(* CODESYS project Raspberry I2C MUX.library
   Author: Stefan Dreyer
   Version: 1.0.1.1
   Description: Library containing device support for different I2C slaves under Raspberry Pi with multiplexer Support
      
      Using some cool function of OSCAT library.
      look at www.oscat.de
   Title: Raspberry I2C MUX
   DefaultNamespace: I2C_MUX
   Company: Stefan Dreyer

Project tree, tasks and I/O mapping:
  libraries: IoStandard, * (System); Standard, * (System); Time and Date, 3.5.7.0 (3S - Smart Software Solutions GmbH); BUILDING, 1.0.0.0 (OSCAT); VisuDialogs, * (System); BASIC, 3.3.3.0 (OSCAT); CAA Memory, 3.5.12.0 (CAA Technical Workgroup); Common Helper for development, 1.0.0.0 (Stefan Dreyer); Raspberry Pi Peripherals, 3.5.13.0 (3S - Smart Software Solutions GmbH); SysSem, 3.5.15.0 (System)
  00000000-0000-0000-0000-000000000000|D:\CoDeSys\LibrariesV3\trunk\Intern\CAA\CAA Template\3.4.0.0 draft\Placeholder.xml
  00000000-0000-0000-0000-000000000000|D:\CoDeSys\LibrariesV3\trunk\Intern\CAA\CAA Template\3.2.0.3 draft\Prefix.pdf
  00000000-0000-0000-0000-000000000000|D:\CoDeSys\LibrariesV3\trunk\Intern\CAA\CAA Template\3.5.2.0 draft\Placeholder.xml
  global variables GVL
  Externe Datei
  Structs/
    data type BusCycleTime
    data type requestData
    data type BME280Data
    data type MUX_COM
    data type SOFT_FONT_DATA
    data type SI7021Data
    data type BMP280Data
  GlobalConstants/
    global variables MyConstants
  Function Blocks/
    function block TCA9548 [ST]: Initialize, BeforeWriteOutputs, goError, BIT_OF_BYTE, restartBus, checkRequestChange, getFirstDifferentStage, clearUnnededStages, setStages
    function block PCA9555OUT [ST]: Initialize, BeforeWriteOutputs
    function block PCA9555IN [ST]: Initialize, AfterReadInputs
    function block BME280 [ST]: AfterReadInputs, Initialize, BeforeWriteOutputs, initCalibration, initDevice, setForcedMode, calcControlRegister
    function block I2C_BASE [ST]: Initialize, AfterReadInputs, BeforeWriteOutputs, checkWrite, checkWrite8, checkReadRegister, goError, checkMultiplex, resetSysCallNum, checkWriteTimeMultiplex, checkReadTimeMultiplex, checkInitMultiplex, checkSet, setRequest, checkMasterFree, resetRequest, checkDeviceOnError, calcCycleTime, checkRead, DeviceState, DeviceRunning
    function block TSL2561 [ST]: AfterReadInputs, Initialize, BeforeWriteOutputs, initDevice, checkDevice, writeControlRegister, setCommandRegister, startDevice, stopDevice, getData, calculateLux
    function block PCF8575IN [ST]: Initialize, AfterReadInputs
    function block PCA9685 [ST]: BeforeWriteOutputs, Initialize, calcOut
    function block Dim4Ch [ST]: BeforeWriteOutputs, Initialize, calcOut
    function block EEPROM_24C512 [ST]: Initialize, AfterReadInputs, BeforeWriteOutputs
    function block SSD1306 [ST]: Initialize, BeforeWriteOutputs, DisplayOn, DisplayOff, SetCommand, SetContrast, DrawLine, SetPixelCache, GetCacheByte, SetCacheByteRaw, WriteCacheToLcd, SetByteCache, SetSoftFont, WriteChar, FillBox, LineFeed, SetCursor
    function block PCF8575OUT [ST]: Initialize, BeforeWriteOutputs
    function block SI7021 [ST]: AfterReadInputs, BeforeWriteOutputs, Initialize
    function block BMP280 [ST]: AfterReadInputs, Initialize, BeforeWriteOutputs, initCalibration, initDevice, setForcedMode, calcControlRegister
  VISU/
    visualisation SSD1306
  text list GlobalTextList
  ENUMS/
    data type LCD_MODES
    data type SOFT_FONT_NUMS
  TextLists/
    text list SOFT_FONT_NAMES
*)

// Structs/BusCycleTime
TYPE BusCycleTime :
STRUCT
	//Cycle Time in ms
	cycleTime:UDINT;
	//last tick for cycle Time
	cycleTimeLastTick:CAA.TICK;
	//cycle frequency 
	cycleFrequency:LREAL;
END_STRUCT
END_TYPE

// Structs/requestData
TYPE requestData :
STRUCT
	//time to next acions
	varTime: CAA.TICK;
	//request var by child outside time, only internal use
	varRequest: BOOL;
	//time between actions in ms
	timePreset:UDINT;
	//set to request by child
	request : BOOL := FALSE;
	//cycle Time of this request
	cycleTime:BusCycleTime;
END_STRUCT
END_TYPE

// Structs/BME280Data
TYPE BME280Data :
STRUCT
	//Possible Data from BME280 from Bosch Sensor Tec
	//using -->LREAL;
	Temperatur:LREAL;//using -->LREAL;
	//using -->LREAL;
	Humidity:LREAL;//using -->LREAL;
	//using -->LREAL;
	Pressure: LREAL;//using -->LREAL;
	//using -->REAL;
	absHumidity:REAL;//using -->REAL;
	//using -->REAL;
	dewPoint:REAL;//using -->REAL;

	(*
		//using -->LREAL;
	Temperatur:CommonTypes.ALL_TYPES_UNION;//using -->LREAL;
	//using -->LREAL;
	Humidity:CommonTypes.ALL_TYPES_UNION;//using -->LREAL;
	//using -->LREAL;
	Pressure: CommonTypes.ALL_TYPES_UNION;//using -->LREAL;
	//using -->REAL;
	absHumidity:CommonTypes.ALL_TYPES_UNION;//using -->REAL;
	//using -->REAL;
	dewPoint:CommonTypes.ALL_TYPES_UNION;//using -->REAL
	*)
	
END_STRUCT
END_TYPE

// Structs/MUX_COM
TYPE MUX_COM :
STRUCT
	
	//Call Number, Order by system call
	callNum:UINT:=0;
	//Start Read differenz for unload cycle load
	//startReadDifferenz:UDINT;
	//muxNum of which slave multiplexer is dead
	//muxNumDead:INT;
	//set this to restart the bus
	startRestartBus: BOOL;

	//set when "last" multiplexer detect to restart the bus
	restartBus: BOOL;
	

	//is init after multiplexer error, all multiplex slaves have to be off
	initAfterError: BOOL;
	//multiplex numbers requestet by on slave
	muxChannelRequest:ARRAY[0..7] OF USINT;
	//multiplex numbers set by master
	muxChannelSet:ARRAY[0..7] OF USINT;
	//instans number of fb who requestet the bus
	fbRequest: INT;

	//count of stages
	stages:UINT;
	//if set, value in stages is valid, so slaves can check there mux nums
	stagesValid: BOOL;
	//mux chain i.O.
	//chainIo:BOOL;
END_STRUCT
END_TYPE

// ENUMS/LCD_MODES
{attribute 'qualified_only'}
{attribute 'strict'}
TYPE LCD_MODES :
(
	CLEAR_BIT := 0, SET_BIT := 1, INVERT_BIT := 2 
)USINT;
END_TYPE

// ENUMS/SOFT_FONT_NUMS
{attribute 'qualified_only'}
{attribute 'strict'}
TYPE SOFT_FONT_NUMS :
(
	FONT_4X6 := 0, FONT_5X8 := 1, FONT_5X12 := 2, FONT_6X8 := 3, FONT_6X10 := 4, FONT_7X12 := 5,
	FONT_7X12B := 6, FONT_8X8 := 7, FONT_8X12 := 8, FONT_8X14 := 9,
	FONT_10X16 := 10, FONT_12X16 := 11, FONT_16X8 := 12,
	FONT_16X12 := 13, FONT_16X26 := 14, last := 15
)USINT;
END_TYPE

// Structs/SOFT_FONT_DATA
TYPE SOFT_FONT_DATA :
STRUCT
	width:USINT;
	height:USINT;
	mask:DWORD;
	data:POINTER TO BYTE;
	size:USINT;
END_STRUCT
END_TYPE

// Structs/SI7021Data
TYPE SI7021Data :
STRUCT
	//Possible Data from BME280 from Bosch Sensor Tec
	//using -->LREAL;
	Temperatur:LREAL;//using -->LREAL;
	//using -->LREAL;
	Humidity:LREAL;//using -->LREAL;
	//using -->REAL;
	absHumidity:REAL;//using -->REAL;
	//using -->REAL;
	dewPoint:REAL;//using -->REAL;

END_STRUCT
END_TYPE

// Structs/BMP280Data
TYPE BMP280Data :
STRUCT
	//Possible Data from BME280 from Bosch Sensor Tec
	//using -->LREAL;
	Temperatur:LREAL;//using -->LREAL;
	//using -->LREAL;
	Pressure: LREAL;//using -->LREAL;

	
END_STRUCT
END_TYPE

// GVL
{attribute 'qualified_only'}
VAR_GLOBAL
	MUX_COMS:ARRAY[0..7]OF MUX_COM;

END_VAR
VAR_GLOBAL CONSTANT
	PCA9685_MODE1: USINT := 0;
	PCA9685_MODE2: USINT := 1;
	PCA9685_PRESCALE: USINT := 16#FE;
	
	LED0_ON_L: USINT := 16#6;
	LED0_ON_H: USINT := 16#7;
	LED0_OFF_L: USINT := 16#8;
	LED0_OFF_H: USINT := 16#9;
END_VAR

// GlobalConstants/MyConstants
{attribute 'qualified_only'}
VAR_GLOBAL CONSTANT

				
END_VAR

// Function Blocks/TCA9548

(*
Function for i2c Multiplexer
so all new, yeha!!!
the slave are requesting an connection to there hardware and writing the channel numbers(of TCA9548) corospending on the hardware in the request array.
and so the master trys to deliver. he checks if a part of the request is already suitable and changes the rest if not.
on init the master tells the slaves how much stages ar avalibel, and so the the slave can check if there config is i.O.
if there are to much stages in the config, the slaves go in error(TODO!!!)
convention: a slave doesn't set a request if the actuel Multiplex set suits his communication request also partially
*)
FUNCTION_BLOCK TCA9548 EXTENDS I2C_BASE

VAR

	stageAddresses:ARRAY[0..7] OF USINT;
	//count of vailid stages
	stages:UINT;
	//which stage ist the last actually
	actLastStage:INT;
	
	outMask:ARRAY[0..7] OF BYTE := [2#1, 2#10, 2#100, 2#1000, 2#10000, 2#100000, 2#1000000, 2#10000000];
	
	//how often i have to try bevor i know i am dead
	retryCountPreload:UINT;
	//var for count trying
	retryCount:UINT;
END_VAR

VAR CONSTANT 
	DEAD_DEVICE:INT:=100;
END_VAR

SUPER^();

METHOD Initialize : UDINT
VAR_INPUT
	wModuleType : UINT;
	dwInstance : UDINT;
	pConnector : POINTER TO IoConfigConnector;
END_VAR
VAR
	pParam: POINTER TO IoConfigParameter;		
	udiResult: UDINT;
 	i:INT;
	iPointer:POINTER TO usINT;
	pLength:DWORD;
END_VAR
SUPER^.Initialize(wModuleType, dwInstance, pConnector);


pParam := ConfigGetParameter(_pConnector, 20);
retryCountPreload := IoStandard.ConfigGetParameterValueWord(pParam, ADR(udiResult));

pParam := ConfigGetParameter(_pConnector, 21);
iPointer := IoStandard.ConfigGetParameterValuePointer(pParam, ADR(udiResult)); 
pLength := IoStandard.ConfigGetParameterLength(pParam);

//copy addresses to instance var
FOR i := 0 TO DWORD_TO_INT(pLength) / 8 DO
	stageAddresses[i+1] := iPointer[i];
END_FOR
//set first stage address in array
stageAddresses[0] := usiAddress;
pParam := ConfigGetParameter(_pConnector, 22);
stages := IoStandard.ConfigGetParameterValueWord(pParam, ADR(udiResult));
GVL.MUX_COMS[numMuxMaster].stages := stages;

GVL.MUX_COMS[numMuxMaster].stagesValid := TRUE;

//actLastStage := 1;

stateAfterError := RETRY_DEVICE;
stateAfterInit := RUN_DEVICE;
//don't use step ERROR_DEVICE in super FB
stateOnError := RETRY_DEVICE;
//GVL.MUX_COMS[numMuxMaster].chainIo := TRUE;
END_METHOD

METHOD BeforeWriteOutputs : INT
VAR
	firstDifferentStage: INT;
	returnByte: BYTE;
END_VAR
SUPER^.BeforeWriteOutputs();

CASE _iState OF

	RUN_DEVICE:
	//hello again folks! i am glad to see you on my next experiment
	//Multiplexing I2C with request from slaves, so lets do it
	IF checkRequestChange() THEN//gotcha, something to do...
		firstDifferentStage := getFirstDifferentStage();
		//if first different in request = 0 then the set have to be resetet from aktStage to Stage 1
		//stage 0 don't need to be cleard, because it is overriden 
		IF actLastStage > firstDifferentStage THEN
			IF clearUnnededStages(firstDifferentStage) = ERROR_RET_VAL THEN
				//error on clear multiplexer
				RETURN;
			END_IF
		END_IF
		IF setStages(firstDifferentStage)  = ERROR_RET_VAL THEN
			RETURN;
		END_IF
	END_IF
 	GVL.MUX_COMS[numMuxMaster].initAfterError := FALSE;
	RETRY_DEVICE:
	IF checkRead(pbyBuffer:= ADR(returnByte), nBufferLen:= 1)  = READ_SUCCSESSFULL THEN
		_iState := RUN_DEVICE;
	END_IF
	//GVL.MUX_COMS[numMuxMaster].chainIo := TRUE;
	
	DEAD_DEVICE:
	//here we can do just nothing ...
	//or wait for an restart from main cycle ...

END_CASE
END_METHOD

METHOD goError
VAR_INPUT
	ReadWrite:BOOL;
END_VAR
VAR
	i:INT;
END_VAR
IF _iState = RUN_DEVICE THEN
	retryCount := retryCountPreload;
END_IF
SUPER^.goError(ReadWrite := FALSE);

//GVL.MUX_COMS[numMuxMaster].chainIo := FALSE;
GVL.MUX_COMS[numMuxMaster].initAfterError := TRUE;
//reset all requests and stages
FOR i := 0 TO  STAGES_END DO
	GVL.MUX_COMS[numMuxMaster].muxChannelSet[i]:= 0;
	GVL.MUX_COMS[numMuxMaster].muxChannelRequest[i]:=0;
END_FOR
END_METHOD

METHOD BIT_OF_BYTE : bool
VAR_INPUT

	in : BYTE;
	N : INT;

END_VAR
BIT_OF_BYTE := (SHR(in,N) AND 16#00000001) > 0;
END_METHOD

//call this from main PUO for try to restart the bus
METHOD restartBus
VAR_INPUT


END_VAR
GVL.MUX_COMS[numMuxMaster].startRestartBus := TRUE;
END_METHOD

METHOD checkRequestChange : bool
VAR_INPUT
END_VAR
VAR
	i:uINT;
END_VAR
//checking if the master have something to to...
checkRequestChange := FALSE;
FOR i := 0 TO stages DO
	IF GVL.MUX_COMS[numMuxMaster].muxChannelRequest[i] <> 0 THEN
		checkRequestChange := TRUE;
	END_IF
END_FOR
END_METHOD

METHOD getFirstDifferentStage : int
VAR_INPUT
END_VAR
VAR
	i:int;	
END_VAR
getFirstDifferentStage := 0;

FOR i := 0 TO 7 DO
	IF GVL.MUX_COMS[numMuxMaster].muxChannelRequest[i] <> GVL.MUX_COMS[numMuxMaster].muxChannelSet[i] THEN
		//it have to hit at interation 7 else a slvae has set an request 
		//for an excisting set
		getFirstDifferentStage := i;
		RETURN;
	END_IF
END_FOR
END_METHOD

METHOD clearUnnededStages : INT
VAR_INPUT
	firstDifferentStage:INT;
	
END_VAR
VAR
	byteBuffer:ARRAY[0..0] OF BYTE;
	i:INT;
	writeRetVal:DINT;
END_VAR
clearUnnededStages := WRITE_SUCCSESSFULL;
//my clear byte
byteBuffer[0] := 0;
FOR i := actLastStage TO firstDifferentStage + 1 BY -1  DO
	//write here with master write
	writeRetVal := _pMaster^.write(stageAddresses[i],ADR(byteBuffer),1);
	IF writeRetVal <> 1 AND NOT debugSlave THEN
		//SUPER^.goError();
		goError(ReadWrite := FALSE);
		clearUnnededStages := ERROR_RET_VAL;
		RETURN;  
	END_IF
	//did go one stage back
	actLastStage := i - 1;
	//and set set
	GVL.MUX_COMS[numMuxMaster].muxChannelSet[i] := 0;
END_FOR
END_METHOD

METHOD setStages : int
VAR_INPUT
	firstDifferentStage:INT;
END_VAR
VAR
	i:INT;
	writeRetVal: DINT;
	byteBuffer: array[0..0] of byte;
END_VAR
setStages := WRITE_SUCCSESSFULL;
FOR i := firstDifferentStage TO 7 DO
	IF GVL.MUX_COMS[numMuxMaster].muxChannelRequest[i] = 0 THEN
		RETURN;//everything done
	END_IF
	byteBuffer[0] := outMask[GVL.MUX_COMS[numMuxMaster].muxChannelRequest[i]-1];
	writeRetVal := _pMaster^.write(stageAddresses[i],ADR(byteBuffer),1);
	IF writeRetVal <> 1 AND NOT debugSlave THEN
		//SUPER^.goError();
		goError(ReadWrite := FALSE);
		setStages := ERROR_RET_VAL;
		RETURN;  
	END_IF
	//set stage set
	GVL.MUX_COMS[numMuxMaster].muxChannelSet[i] := GVL.MUX_COMS[numMuxMaster].muxChannelRequest[i];
	//did go one stage forward
	actLastStage := i;
END_FOR
END_METHOD

END_FUNCTION_BLOCK

// Function Blocks/I2C_BASE
(*Multiplex howto

one I2C_BASE FB is createt by an derive of 3s class i2c

in this fb all Multiplex stuff an controlling Stuff of an i2c slave is beeing done.

childs of this base FB must call parent methods, if theys use and hide the parent method.

the Multiplexing is Programmend for an TCA9548 chip,

you can combinie this chips until the adresses are empty... 

so you can cascade them, or use 8 of them parallel

or 4 parallel an cascade after them, just take care that the adresses can't collid.

in the device descripten the option MUX_MASTER calls the slave behinde which slave they are. It allthow tells the muxer which "row" he serves.

If you cascade the Muxers you don't need to da them in the device tree. the first muxer programm does the stuff for the cascaded ones. so you have to tell the first muxer in the device description,

on which stage after him which adress auf the muxers is being used

So this might an bit confusing, but i did it so ...

So every slave behind an muxer have to tell the master behind which channes of the muxer(s) he is, if he want to communicate.

So you have to see which slaves you do far behinde the pi, because the shold communicate least.

If you have some IO which have to be fast, put them near to the pi

If you have may an io expander with 8 adressesw free, put them behinde one muxer an you can use 8*8 = 64 aof them. ist they are 16 bit then it is 1024 io's

Else, put 8 muxer behinde one muxer and you have 8*8*8*16=8192 IOs. and this with only 9 muxers :D. and 512 IO chips ...

So take care how often the muxed slaves want to communicate because each time the muxer have to be switched.

Allthow you can tell the slaves that they can use foreign requests. This means, if the ar 3 devices behinde on mux channel(don't care aboute the position in the row) and one does request an communication,

The slaves with activatet foreign request do allthow communicatet an reset here own timer. So you can reduse the muxing switching bus load.

You althow cann tell the salve how often they have to communicate, do this in the device description, an look to the exampel devices. 

You althow can request an communication without the timer. Maybe on if an output have changed or you recived an interrupt for an I2C slave.

Look to dhe devices i have used it a some times.

Hi Zdenko,

you need to change this in:

/etc/init.d/codesyscontrol 

snippet:

Code:

        make_mknod

        killall codesyscontrol.bin > /dev/null;

        export PlcConfigFile=/etc/CODESYSControl.cfg

        echo bcm2708_i2c.0 > /sys/bus/platform/drivers/bcm2708_i2c/unbind
        echo 400000 > /sys/module/i2c_bcm2708/parameters/baudrate
        echo bcm2708_i2c.0 > /sys/bus/platform/drivers/bcm2708_i2c/bind




*)
FUNCTION_BLOCK I2C_BASE EXTENDS i2c
VAR_IN_OUT
	
END_VAR

VAR_OUTPUT

	RETVAL:DINT;
	ERROR: BOOL;
	TimeOutHit:BOOL;

END_VAR
VAR
	i:UINT;
	//slave is behind an multiplexer
	isMultiplex: BOOL;
	
 	stageChannelNums:ARRAY[0..STAGES_END] OF USINT;
	//if set use a foreign request to communicate
	useForeign: BOOL;
	//set if an request is set by myself for read
	//requestRead: BOOL;
	//set if an request is set by myself for write
	//requestWrite: BOOL;

	//state auf state maschine after an erre, change on your needs in initialisize
	stateAfterError:INT:=START_INIT;
	stateAfterInit:INT:=START_INIT;
	stateOnError:INT := ERROR_DEVICE;
	
	countNextTry:UDINT;

	waitAfterFault: BOOL;
	cyclseToWaitAfterFault:UDINT:=100;
	
	errorFromChild: BOOL := FALSE;
	

	// Call Number in Order of System call
	sysCallNumRead: UINT;
	sysCallNumWrite: UINT;
	
	readAttempts:LINT;
	writeAttempts:LINT;
	//is Read function called?
	didRead: BOOL := FALSE;
	//is write fucntion called?
	didWrite: BOOL := FALSE;
	//have i to report device i.o.?
	debugSlave: BOOL;
	//request data for read
	readRequest:requestData;
 	//request data for write
	writeRequest:requestData;
	
	numMuxMaster:USINT;
 
	ErrorCountRead:ULINT;
	ErrorCountWrite:ULINT;
	TimeOut:ton;

	
END_VAR
VAR_TEMP	

END_VAR

VAR CONSTANT 

STAGES_END:INT:=7;	

ERROR_DEVICE:INT:=40;
ERROR_RET_VAL:INT:=-1;
WRITE_SUCCSESSFULL:INT:=1;
READ_SUCCSESSFULL:INT:=2;
CHECK_SET_IO:INT:=1;

START_INIT:INT:=5;
WAIT_FOR_STAGES:INT:=1;
START_DEVICE:INT:=6;
RUN_DEVICE:INT:=10;
RETRY_DEVICE:INT:=20;
WAIT_DEVICE:INT:=30;

END_VAR

SUPER^();

(*
try to call this only once per cycle
but it is called by AfterReadInputs an BeforWriteOutputs
so try to check if both function are called by device description 
and if both activ do at read and else in the function called allone

*)
TimeOut(IN := _iState <> 10, PT:=T#1S, Q=> TimeOutHit);

IF _xAfterReadInputs = FALSE AND didRead AND didWrite THEN
	RETURN;
END_IF

//check if mux master gone erre, if so, go self to error
IF checkInitMultiplex() THEN
	goError(ReadWrite := TRUE);
END_IF
 

CASE _iState OF
0:
	IF isMultiplex THEN
		_iState := WAIT_FOR_STAGES;
	ELSE
		_iState := stateAfterInit;
	END_IF
WAIT_FOR_STAGES:
	IF GVL.MUX_COMS[numMuxMaster].stagesValid THEN
		//check muxnums deap
		//if to much muxnums ... error
		FOR i := 0 TO INT_TO_UINT(STAGES_END) DO
			IF stageChannelNums[i] <> 0 AND GVL.MUX_COMS[numMuxMaster].stages < i THEN
				_iState := WAIT_DEVICE;
				
				RETURN;
			END_IF
		END_FOR
		_iState := stateAfterInit;
	END_IF

ERROR_DEVICE:
	IF NOT waitAfterFault THEN
		_iState := stateAfterError;
	ELSE
		IF countNextTry > 0 THEN
			countNextTry := countNextTry- 1;
		END_IF
		IF countNextTry = 0 THEN
			_iState := stateAfterError;
		END_IF
	END_IF
WAIT_DEVICE:
//wrong config, nothing to do
END_CASE


ERROR := _iState <> RUN_DEVICE OR errorFromChild;

METHOD Initialize : UDINT
VAR_INPUT
	wModuleType : UINT;
	dwInstance : UDINT;
	pConnector : POINTER TO IoConfigConnector;
END_VAR
VAR
	pParam: POINTER TO IoConfigParameter;		
	udiResult: UDINT;
	byte1:byte;
	siPointer: POINTER TO USINT;
	pLength: DWORD;
	i: INT;
END_VAR
SUPER^.Initialize(wModuleType, dwInstance, pConnector);
//make differez in start reading, very rudimentary

//MUX_COM.startReadDifferenz := MUX_COM.startReadDifferenz +1;

(*get Adress from config*)
pParam := ConfigGetParameter(_pConnector, 1);
usiAddress:= IoStandard.ConfigGetParameterValueByte(pParam, ADR(udiResult));


(*get status of is this Mutiplex adress*)
pParam := ConfigGetParameter(_pConnector, 2);
byte1:= IoStandard.ConfigGetParameterValueByte(pParam, ADR(udiResult));
IF byte1 = BYTE#1 THEN
	isMultiplex:=TRUE;
ELSE
	isMultiplex:=FALSE;	
END_IF


pParam := ConfigGetParameter(_pConnector, 3);
siPointer := IoStandard.ConfigGetParameterValuePointer(pParam, ADR(udiResult)); 
pLength := IoStandard.ConfigGetParameterLength(pParam);

//copy stages to instance var
FOR i := 0 TO (DWORD_TO_INT(pLength) / 8) DO
	stageChannelNums[i] := siPointer[i];
END_FOR


pParam := ConfigGetParameter(_pConnector, 4);
byte1:= IoStandard.ConfigGetParameterValueByte(pParam, ADR(udiResult));

IF byte1 = BYTE#1 THEN
	waitAfterFault:=TRUE;
ELSE
	waitAfterFault:=FALSE;	
END_IF

pParam := ConfigGetParameter(_pConnector, 5);
cyclseToWaitAfterFault:= IoStandard.ConfigGetParameterValueDword(pParam, ADR(udiResult));

pParam := ConfigGetParameter(_pConnector, 6);
writeRequest.timePreset := IoStandard.ConfigGetParameterValueDword(pParam, ADR(udiResult));



pParam := ConfigGetParameter(_pConnector, 7);
readRequest.timePreset := IoStandard.ConfigGetParameterValueDword(pParam, ADR(udiResult));


pParam := ConfigGetParameter(_pConnector, 8);
byte1:= IoStandard.ConfigGetParameterValueByte(pParam, ADR(udiResult));
IF byte1 = BYTE#1 THEN
	debugSlave:=TRUE;
ELSE
	debugSlave:=FALSE;	
END_IF


pParam := ConfigGetParameter(_pConnector, 9);
byte1:= IoStandard.ConfigGetParameterValueByte(pParam, ADR(udiResult));
IF byte1 = BYTE#1 THEN
	useForeign:=TRUE;
ELSE
	useForeign:=FALSE;	
END_IF
//get mux Master number
pParam := ConfigGetParameter(_pConnector, 10);
numMuxMaster:= IoStandard.ConfigGetParameterValueByte(pParam, ADR(udiResult));
END_METHOD

METHOD AfterReadInputs : INT
VAR
	tick:CAA.TICK;
END_VAR
didRead := TRUE;
SUPER^.AfterReadInputs();

sysCallNumRead := GVL.MUX_COMS[numMuxMaster].callNum;
GVL.MUX_COMS[numMuxMaster].callNum := GVL.MUX_COMS[numMuxMaster].callNum +1;//count to next
END_METHOD

METHOD BeforeWriteOutputs : INT
VAR
	tick: CAA.TICK;
END_VAR
didWrite := TRUE;
SUPER^.BeforeWriteOutputs();


sysCallNumWrite := GVL.MUX_COMS[numMuxMaster].callNum;
GVL.MUX_COMS[numMuxMaster].callNum := GVL.MUX_COMS[numMuxMaster].callNum +1;//count to next
END_METHOD

METHOD checkWrite : INT
VAR_INPUT
	pbyBuffer:POINTER TO BYTE;
	nBufferLen:UDINT;
END_VAR
VAR

END_VAR
IF write(pbyBuffer, nBufferLen) <> UDINT_TO_DINT(nBufferLen) AND NOT debugSlave THEN
	goError(ReadWrite := false);
	checkWrite:=ERROR_RET_VAL;
ELSE
	checkWrite:=WRITE_SUCCSESSFULL;
END_IF
END_METHOD

METHOD checkWrite8 : INT
VAR_INPUT
	usiRegister:USINT;
	usiValue:USINT;
END_VAR
VAR

END_VAR
IF write8(usiRegister, usiValue) = FALSE  AND NOT debugSlave THEN
	goError(ReadWrite := FALSE);
	checkWrite8:=ERROR_RET_VAL;
ELSE
	checkWrite8:=WRITE_SUCCSESSFULL;
END_IF
END_METHOD

METHOD checkReadRegister : INT
VAR_INPUT
	usiRegister:USINT;
	pbyBuffer:POINTER TO BYTE;
	nBufferLen:UDINT;
END_VAR
VAR
	bytesReaded:DINT;
END_VAR
IF readregister(usiRegister, pbyBuffer, nBufferLen) <> UDINT_TO_DINT(nBufferLen) AND NOT debugSlave  THEN //read not suchsseccfull
	goError(ReadWrite := TRUE);
	checkReadRegister := ERROR_RET_VAL;
ELSE
	checkReadRegister := READ_SUCCSESSFULL;
END_IF
END_METHOD

METHOD goError
VAR_INPUT
	//True for read false for write
	ReadWrite:BOOL;
END_VAR
_iState := stateOnError;//Error on accsses 
IF waitAfterFault THEN
	countNextTry := cyclseToWaitAfterFault;
END_IF 
readRequest.varRequest := FALSE;
readRequest.request := FALSE;
writeRequest.varRequest := FALSE;
writeRequest.request := FALSE;

IF ReadWrite THEN

	ErrorCountRead := ErrorCountRead + 1;

ELSE	

	ErrorCountWrite := ErrorCountWrite + 1;

END_IF
END_METHOD

METHOD checkMultiplex : BOOL
VAR_INPUT

	request:POINTER TO requestData;
 
END_VAR
VAR
	checkSetLokal: INT;

END_VAR
checkMultiplex := FALSE;
checkSetLokal := checkSet();

IF request^.timePreset = 0 OR request^.request THEN
	//do here my stuff if i have to read as much as possible
	//or if there is a request by child
	//reset request by child
	//don't check foreign  if we ne can comnunicate 
	//IF checkSetLokal = CHECK_SET_IO AND useForeign THEN
	IF checkSetLokal = CHECK_SET_IO THEN
	//IF checkSetLokal = CHECK_SET_IO THEN
		//if i did the request, delete it
		IF request^.varRequest THEN
			resetRequest(who := ADR(request^.varRequest));
		END_IF
		checkMultiplex := TRUE;
		request^.request := FALSE; 
		RETURN;
	END_IF
	IF NOT request^.varRequest AND checkMasterFree() THEN
		setRequest(who := ADR(request^.varRequest)); // varRequest	
	END_IF
	
ELSE
	//Check if autocycle is disabled
	IF request^.timePreset = 16#FFFFFFFF THEN RETURN; END_IF
	//here do my stuff if i have to wait a few times
	IF checkSetLokal = CHECK_SET_IO AND useForeign AND NOT request^.varRequest THEN
		//on the bus without request and with enabled use foreign request
		//don't do this if i have set an request
		checkMultiplex := TRUE;
		request^.varTime := request^.timePreset + TICKS.GetTick(xDummy:= TRUE);
		RETURN;
	END_IF	
	//check for request
	IF request^.varTime < TICKS.GetTick(xDummy:= TRUE) AND checkMasterFree() THEN
		//new time
		request^.varTime := request^.timePreset + TICKS.GetTick(xDummy:= TRUE);
		//time over, maybe i am already on the bus
		IF checkSetLokal = CHECK_SET_IO THEN
			checkMultiplex := TRUE;
			RETURN;	
		END_IF
		//set request		
		setRequest(who := ADR(request^.varRequest));
	END_IF
	//check if request is fullfilled
	IF checkSetLokal = CHECK_SET_IO AND request^.varRequest THEN
		//my request has been fullfilled
		resetRequest(who := ADR(request^.varRequest));
		checkMultiplex := TRUE;
	END_IF
END_IF
END_METHOD

ACTION resetSysCallNum:
GVL.MUX_COMS[numMuxMaster].callNum := 0;
END_ACTION

METHOD checkWriteTimeMultiplex : bool
VAR_INPUT
	//request data for read
	writeRequest:POINTER TO requestData;
END_VAR
IF isMultiplex THEN
	checkWriteTimeMultiplex := checkMultiplex(request := writeRequest);
ELSE
	checkWriteTimeMultiplex := TRUE;
	//writeRequest^.request := FALSE;
END_IF
IF checkWriteTimeMultiplex THEN
	calcCycleTime(ADR(writeRequest^.cycleTime));
	writeAttempts := writeAttempts + 1; 
END_IF
END_METHOD

METHOD checkReadTimeMultiplex : bool
VAR_INPUT
	//request data for read
	readRequest:POINTER TO requestData;
 
END_VAR
IF isMultiplex THEN
	checkReadTimeMultiplex := checkMultiplex(request := readRequest);
ELSE
	checkReadTimeMultiplex := TRUE;
END_IF
IF checkReadTimeMultiplex THEN
	calcCycleTime(ADR(readRequest^.cycleTime));
	readAttempts := readAttempts + 1; 
END_IF
END_METHOD

//returns true if BUS inits after an multiplexer fault	 
METHOD checkInitMultiplex : bool
VAR_INPUT
END_VAR
 checkInitMultiplex := GVL.MUX_COMS[numMuxMaster].initAfterError AND isMultiplex;
END_METHOD

(*checks if the set deliverd by the master suits to me*)
METHOD checkSet : int
VAR_INPUT
END_VAR
VAR
	i:INT;	
	
END_VAR
checkSet := CHECK_SET_IO;

i := 0;

WHILE stageChannelNums[i] <> 0 AND i < STAGES_END DO
	IF GVL.MUX_COMS[numMuxMaster].muxChannelSet[i] <> stageChannelNums[i] THEN
		checkSet := ERROR_RET_VAL;
		RETURN;
	END_IF 
	i := i + 1;
END_WHILE
END_METHOD

//set request for communication to master
METHOD setRequest : bool
VAR_INPUT
	who:POINTER TO BOOL;
END_VAR
VAR
	i:int;
END_VAR
FOR i := 0 TO STAGES_END DO
	GVL.MUX_COMS[numMuxMaster].muxChannelRequest[i] := stageChannelNums[i];
END_FOR
who^ := TRUE;
END_METHOD

//checks if master is free for new slave	
METHOD checkMasterFree : bool
VAR_INPUT
END_VAR
checkMasterFree := NOT (GVL.MUX_COMS[numMuxMaster].muxChannelRequest[0] <> 0);
END_METHOD

METHOD resetRequest
VAR_INPUT
	who:POINTER TO BOOL;
END_VAR
VAR
	i:int;
END_VAR
FOR i := 0 TO STAGES_END DO
	GVL.MUX_COMS[numMuxMaster].muxChannelRequest[i] := 0;
END_FOR
who^ := FALSE;
END_METHOD

METHOD checkDeviceOnError : bool
VAR_INPUT
END_VAR
checkDeviceOnError := _iState = stateOnError;
END_METHOD

METHOD calcCycleTime : bool
VAR_INPUT
	cycleTime: POINTER TO BusCycleTime;
END_VAR

VAR
	tick: CAA.TICK;
END_VAR
//calaculate cycle time
tick := TICKS.GetTick(xDummy:= TRUE);
cycleTime^.cycleTime := tick - cycleTime^.cycleTimeLastTick; 
cycleTime^.cycleTimeLastTick := tick;
IF cycleTime^.cycleTime = 0 THEN
	//prevend divid by zero
	cycleTime^.cycleTime := 1;
END_IF
cycleTime^.cycleFrequency := 1/(UDINT_TO_LREAL(cycleTime^.cycleTime)/1000);
calcCycleTime  := TRUE;
END_METHOD

METHOD checkRead : INT
VAR_INPUT
	pbyBuffer:POINTER TO BYTE;
	nBufferLen:UDINT;
END_VAR
IF read(pbyBuffer, nBufferLen) <> UDINT_TO_DINT(nBufferLen) AND NOT debugSlave  THEN //read not suchsseccfull
	goError(ReadWrite := TRUE);
	checkRead := ERROR_RET_VAL;
ELSE
	checkRead := READ_SUCCSESSFULL;
END_IF
END_METHOD

PROPERTY DeviceState : int
GET
DeviceState := _iState;
END_GET
END_PROPERTY

PROPERTY DeviceRunning : bool
GET
DeviceRunning := _iState = RUN_DEVICE;
END_GET
END_PROPERTY

END_FUNCTION_BLOCK

// Function Blocks/PCA9555OUT
FUNCTION_BLOCK PCA9555OUT EXTENDS I2C_BASE
VAR_INPUT
	
	outs: ARRAY[0..1] OF BYTE;
	
END_VAR
VAR
	hiOld:BYTE;
	lowOld:BYTE;
	
END_VAR

SUPER^();

METHOD Initialize : UDINT
VAR_INPUT
	wModuleType : UINT;
	dwInstance : UDINT;
	pConnector : POINTER TO IoConfigConnector;
END_VAR
VAR
	pParam: POINTER TO IoConfigParameter;		
	udiResult: UDINT;
	byte1:byte;
END_VAR
SUPER^.Initialize(wModuleType, dwInstance, pConnector);
END_METHOD

METHOD BeforeWriteOutputs : INT
VAR
	i: USINT;
	pyBuffer:ARRAY[0..2]OF BYTE;
END_VAR
SUPER^.BeforeWriteOutputs();

//GVL.callNum := 0;
IF checkInitMultiplex() THEN
	RETURN;
END_IF
CASE _iState OF
START_DEVICE:
	writeRequest.request := TRUE;
	IF NOT checkWriteTimeMultiplex(ADR(writeRequest)) THEN
		RETURN;
	END_IF 
	checkWrite8(6,0);
	checkWrite8(7,0);
	IF _iState<>ERROR_DEVICE THEN
		_iState := RUN_DEVICE;	
	END_IF
	//write Output, this is for return after error state
	
	IF checkWrite8(2,outs[0]) < 0 THEN
		RETURN ;
	END_IF
	lowOld := outs[0];
	

	IF checkWrite8(3,outs[1]) < 0 THEN
		RETURN ;
	END_IF
	hiOld := outs[1];

RUN_DEVICE:
	//requestWrite
	IF lowOld <> outs[0] OR hiOld <> outs[1] THEN
		writeRequest.request := TRUE;
	END_IF
	IF NOT checkWriteTimeMultiplex(ADR(writeRequest)) THEN
		RETURN;
	END_IF
	//reset request
	writeRequest.request := FALSE;
	//save old values
	lowOld := outs[0];
	hiOld := outs[1];
	//write 2 bytes --> faster
	pyBuffer[0] := 2;
	pyBuffer[1] := outs[0];
	pyBuffer[2] := outs[1];
	checkWrite(ADR(pyBuffer),3);
	
END_CASE
END_METHOD

END_FUNCTION_BLOCK

// Function Blocks/PCA9555IN
FUNCTION_BLOCK PCA9555IN EXTENDS I2C_BASE

VAR_OUTPUT
	ins: ARRAY[0..1] OF BYTE;
END_VAR

SUPER^();

METHOD Initialize : UDINT
VAR_INPUT
	wModuleType : UINT;
	dwInstance : UDINT;
	pConnector : POINTER TO IoConfigConnector;
END_VAR
VAR

END_VAR
SUPER^.Initialize(wModuleType, dwInstance, pConnector);


stateAfterError := RUN_DEVICE;
stateAfterInit := RUN_DEVICE;
END_METHOD

METHOD AfterReadInputs : INT
VAR

END_VAR
SUPER^.AfterReadInputs();

IF checkInitMultiplex() THEN
	RETURN;
END_IF

CASE _iState OF

RUN_DEVICE:
	//check if time are over
	IF NOT checkReadTimeMultiplex(ADR(readRequest)) THEN
		RETURN;
	END_IF
	checkReadRegister(16#0,ADR(ins),2);
	
END_CASE
END_METHOD

END_FUNCTION_BLOCK

// Function Blocks/BME280
FUNCTION_BLOCK BME280 EXTENDS I2C_BASE
VAR_INPUT

END_VAR
VAR_OUTPUT
	myData:BME280Data;
	configWrong: BOOL;
END_VAR
VAR


	dig_T1: LREAL;
    dig_T2: LREAL;
    dig_T3: LREAL;
	 
    dig_P1: LREAL;
    dig_P2: LREAL;
    dig_P3: LREAL;
    dig_P4: LREAL;
    dig_P5: LREAL;
    dig_P6: LREAL;
    dig_P7: LREAL;
    dig_P8: LREAL;
    dig_P9: LREAL;

    dig_H1: LREAL;
    dig_H2: LREAL;
    dig_H3: LREAL;
    dig_H4: LREAL;
    dig_H5: LREAL;
    dig_H6: LREAL;

	t_fine:DINT;
	
	tempOversampling: USINT;
	pressureOversampling: USINT;
	humidityOversampling: USINT;
	iirFilter:USINT;
	standbyTime:USINT;
	controlRegister:BYTE;
	writeControlRegister:BOOL;
	operationMode:BYTE;
	//diffrenz for read the next value in ms
	nextForcedDiff:UDINT;
	//next time to write forced
	nextForced: CAA.TICK;
	//wrong device!
	wrongDevice: BOOL;


END_VAR
VAR_TEMP	
END_VAR

VAR CONSTANT 
	
BME280_REGISTER_DIG_T1:USINT := 16#88;
BME280_REGISTER_DIG_T2:USINT := 16#8A;
BME280_REGISTER_DIG_T3:USINT := 16#8C;

BME280_REGISTER_DIG_P1:USINT := 16#8E;
BME280_REGISTER_DIG_P2:USINT := 16#90;
BME280_REGISTER_DIG_P3:USINT := 16#92;
BME280_REGISTER_DIG_P4:USINT := 16#94;
BME280_REGISTER_DIG_P5:USINT := 16#96;
BME280_REGISTER_DIG_P6:USINT := 16#98;
BME280_REGISTER_DIG_P7:USINT := 16#9A;
BME280_REGISTER_DIG_P8:USINT := 16#9C;
BME280_REGISTER_DIG_P9:USINT := 16#9E;

BME280_REGISTER_DIG_H1:USINT := 16#A1;
BME280_REGISTER_DIG_H2:USINT := 16#E1;
BME280_REGISTER_DIG_H3:USINT := 16#E3;
BME280_REGISTER_DIG_H4:USINT := 16#E4;
BME280_REGISTER_DIG_H5:USINT := 16#E5;
BME280_REGISTER_DIG_H6:USINT := 16#E6;
BME280_REGISTER_DIG_H7:USINT := 16#E7;	

BME280_REGISTER_CHIPID:USINT := 16#D0;
BME280_REGISTER_VERSION :USINT := 16#D1;
BME280_REGISTER_SOFTRESET :USINT := 16#E0;

BME280_REGISTER_CONTROL_HUM :USINT := 16#F2;
BME280_REGISTER_CONTROL :USINT := 16#F4;
BME280_REGISTER_CONFIG :USINT := 16#F5;
BME280_REGISTER_PRESSURE_DATA :USINT := 16#F7;
BME280_REGISTER_TEMP_DATA :USINT := 16#FA;
BME280_REGISTER_HUMIDITY_DATA :USINT := 16#FD;
BME_280_DEVICE_ID:USINT:=16#60;

TEMP_OVERSAMPLING_MAX:USINT:=5;
PRESSURE_OVERSAMPLING_MAX:USINT:=5;
HUMIDITY_OVERSAMPLING_MAX:USINT:=5;
IIR_FILTER_MAX:USINT:=4;
STANDBY_TIME_MAX:USINT:=7;
BME280_NORMAL_MODE:USINT:=2#11;
BME280_FORCED_MODE:USINT:=2#01;
BME280_SLEEP_MODE:USINT:=2#00;

TEMPERATURE_OFF:UDINT:=16#80000;
PRESSURE_OFF:UDINT:=16#80000;
HUMIDITY_OFF:UDINT:=16#8000;



END_VAR

SUPER^();

CASE _iState OF
	RUN_DEVICE:
		IF operationMode = BME280_FORCED_MODE THEN
			IF nextForced < TICKS.GetTick(xDummy:= TRUE) THEN
				//set next read
				nextForced := nextForcedDiff + TICKS.GetTick(xDummy:= TRUE);
				setForcedMode();
				
			END_IF 
		ELSE
			nextForced := nextForcedDiff + TICKS.GetTick(xDummy:= TRUE);
		END_IF
END_CASE

METHOD AfterReadInputs : INT
VAR
	sensorData: ARRAY[0..7] OF BYTE;	
	rawTempSensor:UDINT;
	rawTemp:LREAL;
	rawPressureSensor:UDINT;
	rawPressure:LREAL;
	rawHumiditySensor:UDINT;
	rawHumidity:LREAL;
	var1, var2, p, var_H:LREAL;
	tError, hError, pError: BOOL;
	//dd:LREAL;
END_VAR
SUPER^.AfterReadInputs();

IF checkInitMultiplex() THEN
	RETURN;
END_IF
CASE _iState OF
START_INIT:
	readRequest.request := TRUE;
	
	//check if time are over
	IF NOT checkReadTimeMultiplex(ADR(readRequest)) THEN
		RETURN;
	END_IF
	initCalibration();

	IF _iState<>ERROR_DEVICE THEN
		_iState := START_DEVICE;

	END_IF
RUN_DEVICE:
	//check if time are over
	IF NOT checkReadTimeMultiplex(ADR(readRequest)) THEN
		RETURN;
	END_IF
	(*read all sensor Data*)
	IF checkReadRegister(BME280_REGISTER_PRESSURE_DATA, ADR(sensorData),8) < 0 THEN
		RETURN;
	END_IF
	
	rawTempSensor:=0;
	rawTempSensor:=SHL(BYTE_TO_UDINT(sensorData[3]),16);
	rawTempSensor:=rawTempSensor OR SHL(BYTE_TO_UDINT(sensorData[4]),8);
	rawTempSensor:=rawTempSensor OR BYTE_TO_UDINT(sensorData[5]);
	rawTempSensor:= SHR(rawTempSensor,4);
	//if Sensor value off and sensor switched on(no power)
	IF rawTempSensor = TEMPERATURE_OFF AND tempOversampling >0 THEN
		goError(ReadWrite := TRUE);
		RETURN;
	END_IF
	IF rawTempSensor <> 16#80000 THEN
		rawTemp:=UDINT_TO_REAL(rawTempSensor);
		var1  := (rawTemp/16384.0 - dig_T1/1024.0) * dig_T2;
		var2  := ((rawTemp/131072.0 - dig_T1/8192.0) *   (rawTemp/131072.0 -  dig_T1/8192.0)) * dig_T3;
		t_fine := LREAL_TO_DINT(var1 + var2);
		myData.Temperatur  := (var1 + var2) / 5120.0;
		
	ELSE
		myData.Temperatur:=0.0;
		
	END_IF
	//Calculate pressure
	rawPressureSensor:=0;
	rawPressureSensor:=SHL(BYTE_TO_UDINT(sensorData[0]),16);
	rawPressureSensor:=rawPressureSensor OR SHL(BYTE_TO_UDINT(sensorData[1]),8);
	rawPressureSensor:=rawPressureSensor OR BYTE_TO_UDINT(sensorData[2]);
	rawPressureSensor:= SHR(rawPressureSensor,4);
	IF rawPressureSensor = PRESSURE_OFF AND pressureOversampling >0 THEN
		goError(ReadWrite := TRUE);
		RETURN;
	END_IF
	IF rawPressureSensor <> 16#80000 THEN
		rawPressure:=UDINT_TO_REAL(rawPressureSensor);
		var1 := (DINT_TO_LREAL(t_fine)/2.0) - 64000.0;
		var2 := var1 * var1 * (dig_P6) / 32768.0;
		var2 := var2 + var1 * (dig_P5) * 2.0;
		var2 := (var2/4.0)+((dig_P4) * 65536.0);
		var1 := ((dig_P3) * var1 * var1 / 524288.0 + (dig_P2) * var1) / 524288.0;
		var1 := (1.0 + var1 / 32768.0)*(dig_P1);
		IF var1 = 0.0 THEN
			myData.Pressure := 0.0;
		ELSE	
			p := 1048576.0 - rawPressure;
			p := (p - (var2 / 4096.0)) * 6250.0 / var1;
			var1 := (dig_P9) * p * p / 2147483648.0;
			var2 := p * (dig_P8) / 32768.0;
			p := p + (var1 + var2 + (dig_P7)) / 16.0;
			myData.Pressure := p; 	
		END_IF
  	ELSE
		myData.Pressure :=0.0;
	END_IF
	//humidity
	
	rawHumiditySensor:=0;
	rawHumiditySensor:=SHL(BYTE_TO_UDINT(sensorData[6]),8);
	rawHumiditySensor:=rawHumiditySensor OR BYTE_TO_UDINT(sensorData[7]);
	IF rawHumiditySensor = HUMIDITY_OFF AND humidityOversampling >0 THEN
		goError(ReadWrite := TRUE);
		RETURN;
	END_IF
	IF rawHumiditySensor <> 16#8000 THEN
		rawHumidity:=UDINT_TO_REAL(rawHumiditySensor);
		var_H := (DINT_TO_LREAL(t_fine) - 76800.0);
		var_H := (rawHumidity - ((dig_H4) * 64.0 + (dig_H5) / 16384.0 * var_H)) * 
			((dig_H2) / 65536.0 * (1.0 + (dig_H6) / 67108864.0 * var_H *  (1.0 + (dig_H3) / 67108864.0 * var_H)));
		var_H := var_H * (1.0 - (dig_H1) * var_H / 524288.0);
		IF var_H > 100.0 THEN
		   var_H := 100.0;
		ELSIF var_H < 0.0 THEN 
		  var_H := 0.0; 
		END_IF
		myData.Humidity :=var_H;
	ELSE
		myData.Humidity :=0.0;
	END_IF
	

	myData.absHumidity  := OSCAT_BUILDING.DEW_CON(RH:=LREAL_TO_REAL(myData.Humidity) , T:=LREAL_TO_REAL(myData.Temperatur) );
	myData.dewPoint := OSCAT_BUILDING.DEW_TEMP(RH:= LREAL_TO_REAL(myData.Humidity), T:=LREAL_TO_REAL(myData.Temperatur ));


	
END_CASE
END_METHOD

METHOD Initialize : UDINT
VAR_INPUT
	wModuleType : UINT;
	dwInstance : UDINT;
	pConnector : POINTER TO IoConfigConnector;
END_VAR
VAR
	pParam: POINTER TO IoConfigParameter;		
	udiResult: UDINT;
	byte1:byte;
END_VAR
SUPER^.Initialize(wModuleType, dwInstance, pConnector);

IF usiAddress = 0 THEN
	usiAddress := 16#77;
END_IF


pParam := ConfigGetParameter(_pConnector, 20);
tempOversampling:= IoStandard.ConfigGetParameterValueByte(pParam, ADR(udiResult));
IF tempOversampling > TEMP_OVERSAMPLING_MAX THEN
	 tempOversampling := TEMP_OVERSAMPLING_MAX;
	configWrong := TRUE; 
END_IF
pParam := ConfigGetParameter(_pConnector, 21);
pressureOversampling:= IoStandard.ConfigGetParameterValueByte(pParam, ADR(udiResult));
IF pressureOversampling > PRESSURE_OVERSAMPLING_MAX THEN
	pressureOversampling := PRESSURE_OVERSAMPLING_MAX;
	configWrong := TRUE;
END_IF
pParam := ConfigGetParameter(_pConnector, 22);
humidityOversampling:= IoStandard.ConfigGetParameterValueByte(pParam, ADR(udiResult));
IF humidityOversampling > HUMIDITY_OVERSAMPLING_MAX THEN
	 humidityOversampling := HUMIDITY_OVERSAMPLING_MAX;
	 configWrong := TRUE;
END_IF
pParam := ConfigGetParameter(_pConnector, 23);
iirFilter:= IoStandard.ConfigGetParameterValueByte(pParam, ADR(udiResult));
IF iirFilter > IIR_FILTER_MAX THEN
	iirFilter := IIR_FILTER_MAX;
	configWrong := TRUE;
END_IF
pParam := ConfigGetParameter(_pConnector, 24);
standbyTime:= IoStandard.ConfigGetParameterValueByte(pParam, ADR(udiResult));
IF standbyTime > STANDBY_TIME_MAX THEN
	standbyTime := STANDBY_TIME_MAX;
	configWrong := TRUE;
END_IF

pParam := ConfigGetParameter(_pConnector, 25);
nextForcedDiff:= IoStandard.ConfigGetParameterValueDWord(pParam, ADR(udiResult));
IF nextForcedDiff = 0  THEN
	operationMode := BME280_NORMAL_MODE;
ELSE
	operationMode := BME280_FORCED_MODE;
END_IF


errorFromChild := configWrong;

stateAfterError := START_INIT;
stateAfterInit := START_INIT;
END_METHOD

METHOD BeforeWriteOutputs : INT
VAR

END_VAR
SUPER^.BeforeWriteOutputs();

IF checkInitMultiplex() THEN
	RETURN;
END_IF

CASE _iState OF
START_DEVICE:
	//check if time is over
	//writeRequest.request := requestOnInit;
	writeRequest.request := TRUE;
	IF checkWriteTimeMultiplex(ADR(writeRequest)) = FALSE  THEN
		RETURN;// i am not on the bus
	END_IF
	
	initDevice();
	IF _iState<>ERROR_DEVICE THEN
		_iState := RUN_DEVICE;
		//requestOnInit := FALSE;//init successful	
	END_IF
	
RUN_DEVICE:
	IF checkWriteTimeMultiplex(ADR(writeRequest)) = FALSE  THEN
		RETURN;// i am not on the bus
	END_IF
	IF writeControlRegister THEN
		IF checkWrite8(BME280_REGISTER_CONTROL,controlRegister) < 0 THEN
			RETURN;
		ELSE
			writeControlRegister := FALSE;
			IF operationMode = BME280_FORCED_MODE THEN
				readRequest.request := TRUE;
			END_IF
		END_IF
	END_IF
	
	
END_CASE
END_METHOD

METHOD initCalibration
VAR_INPUT
END_VAR
VAR
	byte1: BYTE;
	byte2: BYTE;
	x: INT;
	tint:INT;
	tuint:UINT;
	tusint:USINT;
	tsint:SINT;
	
END_VAR
(*read calibration values from BME 280 *)
//check device
IF checkReadRegister(BME280_REGISTER_CHIPID, ADR(tusint),1) < 0 THEN
	RETURN;
END_IF
IF tusint <> BME_280_DEVICE_ID THEN//wrong device --> go error
	goError(ReadWrite:= TRUE);
	wrongDevice := TRUE;
	RETURN;
ELSE
	wrongDevice := FALSE;
END_IF
IF checkReadRegister(BME280_REGISTER_DIG_T1, ADR(tuint),2) < 0 THEN
	RETURN;
END_IF
dig_T1 := UINT_TO_LREAL(tuint);
IF checkReadRegister(BME280_REGISTER_DIG_T2, ADR(tint),2) < 0 THEN
	RETURN;
END_IF 
dig_T2 := INT_TO_LREAL(tint);
IF checkReadRegister(BME280_REGISTER_DIG_T3, ADR(tint),2) < 0 THEN
	RETURN;
END_IF
dig_T3 := INT_TO_LREAL(tint);

IF checkReadRegister(BME280_REGISTER_DIG_P1, ADR(tuint),2) <0 THEN
	RETURN;
END_IF
dig_P1 := UINT_TO_LREAL(tuint);
IF checkReadRegister(BME280_REGISTER_DIG_P2, ADR(tint),2) < 0 THEN
	RETURN;
END_IF
dig_P2 := INT_TO_LREAL(tint);
IF checkReadRegister(BME280_REGISTER_DIG_P3, ADR(tint),2) < 0 THEN
	RETURN;
END_IF
dig_P3 := INT_TO_LREAL(tint);
IF checkReadRegister(BME280_REGISTER_DIG_P4, ADR(tint),2) < 0 THEN
	RETURN;
END_IF
dig_P4 := INT_TO_LREAL(tint);
IF checkReadRegister(BME280_REGISTER_DIG_P5, ADR(tint),2) < 0 THEN
	RETURN;
END_IF
dig_P5 := INT_TO_LREAL(tint);
IF checkReadRegister(BME280_REGISTER_DIG_P6, ADR(tint),2) < 0 THEN
	RETURN;
END_IF
dig_P6 := INT_TO_LREAL(tint);
IF checkReadRegister(BME280_REGISTER_DIG_P7, ADR(tint),2) < 0 THEN
	RETURN;
END_IF
dig_P7 := INT_TO_LREAL(tint);
IF checkReadRegister(BME280_REGISTER_DIG_P8, ADR(tint),2) < 0 THEN
	RETURN;
END_IF
dig_P8 := INT_TO_LREAL(tint);
IF checkReadRegister(BME280_REGISTER_DIG_P9, ADR(tint),2) < 0 THEN
	RETURN;
END_IF
dig_P9 := INT_TO_LREAL(tint);


IF checkReadRegister(BME280_REGISTER_DIG_H1, ADR(tusint),1) < 0 THEN
	RETURN;
END_IF
dig_H1 := USINT_TO_LREAL(tusint);
IF checkReadRegister(BME280_REGISTER_DIG_H2, ADR(tint),2) < 0 THEN
	RETURN;
END_IF
dig_H2 := INT_TO_LREAL(tint);
IF checkReadRegister(BME280_REGISTER_DIG_H3, ADR(tusint),1) < 0 THEN
	RETURN;
END_IF
dig_H3 := USINT_TO_LREAL(tusint);
IF checkReadRegister(BME280_REGISTER_DIG_H7, ADR(tsint),1) < 0 THEN
	RETURN;
END_IF
dig_H6 := SINT_TO_LREAL(tsint);


IF checkReadRegister(BME280_REGISTER_DIG_H4, ADR(BYTE1),1) < 0 THEN
	RETURN;
END_IF
IF checkReadRegister(BME280_REGISTER_DIG_H5, ADR(BYTE2),1) < 0 THEN
	RETURN;
END_IF

dig_H4 := UINT_TO_LREAL(SHL(INT_TO_UINT(BYTE_TO_INT(byte1)),4) OR (byte2 AND 16#0F));
IF checkReadRegister(BME280_REGISTER_DIG_H6, ADR(BYTE1),1) < 0 THEN
	RETURN;
END_IF
dig_H5 := UINT_TO_LREAL(SHL(INT_TO_UINT(BYTE_TO_INT(byte1)),4) OR (SHR(byte2,4) AND 16#0F));
END_METHOD

METHOD initDevice : INT
VAR_INPUT
END_VAR
IF checkWrite8(BME280_REGISTER_CONFIG, (SHL(standbyTime,5)OR SHL(iirFilter,2))) < 0 THEN
	RETURN;		
END_IF
	
IF checkWrite8(BME280_REGISTER_CONTROL_HUM, humidityOversampling) < 0 THEN
	RETURN;
END_IF
	calcControlRegister();
IF checkWrite8(BME280_REGISTER_CONTROL,controlRegister) < 0 THEN
	RETURN;
END_IF
END_METHOD

METHOD setForcedMode
VAR_INPUT
END_VAR
operationMode := BME280_FORCED_MODE;
calcControlRegister();
writeControlRegister := TRUE;
writeRequest.request := TRUE;
END_METHOD

METHOD calcControlRegister
VAR_INPUT
END_VAR
controlRegister := SHL(tempOversampling,5)OR SHL(pressureOversampling,2)OR operationMode;
END_METHOD

END_FUNCTION_BLOCK

// Function Blocks/TSL2561
(*HOWTO
	first set gain to max(16) an then read the sensor
	after that check if AD Value ist to high(sensor is saturated)
	if not, so calc lux value,
	if so set the gain to 1 and the read and calculate 
	we can't use ms between read, because, sometimes we have to read twice for good result,
	so we have an extra parameter for cycle time*)
FUNCTION_BLOCK TSL2561 EXTENDS I2C_BASE
VAR_INPUT
END_VAR
VAR_OUTPUT
	configWrong: BOOL;
END_VAR
VAR
	gain:USINT;
	integrationTime:USINT;
	mySteps:INT := 0;
	waitIntegration : CAA.TICK;
	cycleTime : CAA.TICK;
	cycleTimePreset:UDINT;
	fullData:UINT;
	irData:UINT;
	lux:LREAL;
	//True for CS Package, false for T, FN and CL Package
	package: BOOL;
	//all vars for scaling
	//scale area 1
	scale1CheckHigh:LREAL;
	scale1Calc1:LREAL;
	scale1Calc2:LREAL;
	//scale area 2
	scale2CheckLow:LREAL;
	scale2CheckHigh:LREAL;
	scale2Calc1:LREAL;
	scale2Calc2:LREAL;
	//scale area 3
	scale3CheckLow:LREAL;
	scale3CheckHigh:LREAL;
	scale3Calc1:LREAL;
	scale3Calc2:LREAL;
	//scale area 4
	scale4CheckLow:LREAL;
	scale4CheckHigh:LREAL;
	scale4Calc1:LREAL;
	scale4Calc2:LREAL;
	//scale area 5
	scale5CheckHigh:LREAL;
	
	
END_VAR

VAR CONSTANT
	GAIN_MAX: USINT := 1;
	INTEGRATION_TIME_MAX: USINT := 3;
	
	TSL2561_COMMAND_REGISTER_BIT: USINT := 2#10000000;
	TSL2561_BLOCK_COMMAND: USINT := 2#10000;
	TSL2561_CONTROLL_REGISTER_ADRESS: USINT := 0;
	TSL2561_TIMING_REGISTER_ADRESS: USINT := 16#1;
	TSL2561_SENSOR_REGISTER_ADRESS:USINT := 16#C;
	TSL2561_ID_REGISTER_ADRESS:USINT := 16#A;
	TSL2561_MANUAL_START:USINT:=2#1000;
	TSL2561_DEVICE_START:USINT:=16#3;
	TSL2561_DEVICE_STOP:USINT:=16#0;
	
	TSL2561_GAIN_LOW:USINT:=0;
	TSL2561_GAIN_HIGH:USINT:=1;
	
	TSL2561_INTEGATION_TIME:ARRAY[0..2] OF UINT:=[15,105,405];
	TSL2561_INTEGRATION_TIME_SCALE:ARRAY[0..2]OF LREAL:=[0.034,0.252,1];
	
	TSL2561_INTEGATION_TIME_LOW_SET:USINT:=2#0;
	TSL2561_INTEGATION_TIME_MID_SET:USINT:=2#1;
	TSL2561_INTEGATION_TIME_HIGH_SET:USINT:=2#10;
	TSL2561_INTEGATION_TIME_HIGH_OFF:USINT:=2#11;
	
	TSL2561_GAIN_LIMIT_LOW:UINT:=4000;
	
	//Steps for _iStep
	STEP_CHECK_DEVICE : INT := 1;

	//Steps for myStep
	//STEP_CHANGE_PARAMS: INT := 2;
	//STEP_INIT_DEVICE:INT:=2;
	//STEP_SET_HIGH:INT:=1;
	//STEP_READ_HIGH:INT:=2;
	STEP_READ:INT:=5;
	//STEP_SET_LOW:INT:=3;
	//STEP_READ_LOW:INT:=4;
	STEP_WAIT:INT:=6;
	STEP_START_DEVICE:INT:=7;
END_VAR

SUPER^();

METHOD AfterReadInputs : INT
VAR
END_VAR
SUPER^.AfterReadInputs();

IF checkInitMultiplex() THEN
	RETURN;
END_IF

CASE _iState OF

STEP_CHECK_DEVICE:
	readRequest.request := TRUE;
	IF NOT checkReadTimeMultiplex(ADR(readRequest)) THEN
		RETURN;
	END_IF
	IF checkDevice() = FALSE THEN
		RETURN;
	END_IF
	_iState := START_DEVICE;	

	
RUN_DEVICE:
	CASE mySteps OF
		STEP_READ:
			//wait till integration time is over
			IF waitIntegration >  TICKS.GetTick(xDummy:=TRUE) THEN
				RETURN;
			END_IF
			readRequest.request := TRUE;
			IF NOT checkReadTimeMultiplex(ADR(readRequest)) THEN
				RETURN;
			END_IF
			IF getData() < 0 THEN
				RETURN;
			END_IF
			IF stopDevice() < 0 THEN
				RETURN;
			END_IF
			
			IF gain = TSL2561_GAIN_LOW AND (irData < TSL2561_GAIN_LIMIT_LOW AND fullData < TSL2561_GAIN_LIMIT_LOW) THEN
				gain := TSL2561_GAIN_HIGH;
				mySteps := STEP_START_DEVICE;
				RETURN;
			END_IF
			
			
			IF irData = 16#FFFF OR fullData = 16#FFFF THEN
				//Value(s) exeed(s) datarange, now try low gain
				gain := TSL2561_GAIN_LOW;
				mySteps := STEP_START_DEVICE;
				RETURN;
			END_IF
			//here we can calculate LUX
			calculateLux();
			mySteps := STEP_WAIT;
	
			
		STEP_WAIT:
		IF cycleTime < TICKS.GetTick(xDummy:= TRUE) THEN
			mySteps := STEP_START_DEVICE;
			cycleTime := TICKS.GetTick(xDummy:= TRUE) + cycleTimePreset; 
		END_IF	
	END_CASE
	
RETRY_DEVICE:

	IF checkDevice() = FALSE THEN
		RETURN;
	END_IF
	_iState := START_DEVICE;	

END_CASE
END_METHOD

METHOD Initialize : UDINT
VAR_INPUT
	wModuleType : UINT;
	dwInstance : UDINT;
	pConnector : POINTER TO IoConfigConnector;
END_VAR
VAR
	pParam: POINTER TO IoConfigParameter;		
	udiResult: UDINT;
	byte1:byte;
END_VAR
SUPER^.Initialize(wModuleType, dwInstance, pConnector);

IF usiAddress = 0 THEN
	usiAddress := 16#29;
END_IF
configWrong := FALSE;

pParam := ConfigGetParameter(_pConnector, 20);
byte1:= IoStandard.ConfigGetParameterValueByte(pParam, ADR(udiResult));
IF byte1 = BYTE#1 THEN
	package:=TRUE;
ELSE
	package:=FALSE;	
END_IF


IF package THEN
	//scale area 1
	scale1CheckHigh:=LREAL#0.52;
	scale1Calc1:=LREAL#0.0315;
	scale1Calc2:=LREAL#0.0593;
	//scale area 2
	scale2CheckLow:=LREAL#0.52;
	scale2CheckHigh:=LREAL#0.65;
	scale2Calc1:=LREAL#0.0229;
	scale2Calc2:=LREAL#0.0291;
	//scale area 3
	scale3CheckLow:=LREAL#0.65;
	scale3CheckHigh:=LREAL#0.80;
	scale3Calc1:=LREAL#0.0157;
	scale3Calc2:=LREAL#0.0180;
	//scale area 4
	scale4CheckLow:=LREAL#0.80;
	scale4CheckHigh:=LREAL#0.130;
	scale4Calc1:=LREAL#0.00338;
	scale4Calc2:=LREAL#0.00260;
	//scale area 5
	scale5CheckHigh:=LREAL#1.3;
ELSE
	//scale area 1
	scale1CheckHigh:=LREAL#0.5;
	scale1Calc1:=LREAL#0.0304;
	scale1Calc2:=LREAL#0.062;
	//scale area 2
	scale2CheckLow:=LREAL#0.50;
	scale2CheckHigh:=LREAL#0.61;
	scale2Calc1:=LREAL#0.0224;
	scale2Calc2:=LREAL#0.031;
	//scale area 3
	scale3CheckLow:=LREAL#0.61;
	scale3CheckHigh:=LREAL#0.80;
	scale3Calc1:=LREAL#0.0128;
	scale3Calc2:=LREAL#0.0153;
	//scale area 4
	scale4CheckLow:=LREAL#0.80;
	scale4CheckHigh:=LREAL#1.30;
	scale4Calc1:=LREAL#0.00146;
	scale4Calc2:=LREAL#0.00112;
	//scale area 5
	scale5CheckHigh:=LREAL#1.3;
END_IF

pParam := ConfigGetParameter(_pConnector, 21);
//integrationTime := TSL2561_INTEGATION_TIME_HIGH_OFF;
integrationTime:= IoStandard.ConfigGetParameterValueByte(pParam, ADR(udiResult));
IF integrationTime > INTEGRATION_TIME_MAX THEN
	integrationTime := INTEGRATION_TIME_MAX;
	configWrong := TRUE;
END_IF
//fix integration until we change the calculation
integrationTime := INTEGRATION_TIME_MAX - 1;

pParam := ConfigGetParameter(_pConnector, 22);
cycleTimePreset := IoStandard.ConfigGetParameterValueDword(pParam, ADR(udiResult));

errorFromChild := configWrong;

stateAfterError := RETRY_DEVICE;
stateAfterInit := RETRY_DEVICE;
END_METHOD

METHOD BeforeWriteOutputs : INT
VAR

END_VAR
SUPER^.BeforeWriteOutputs();

IF checkInitMultiplex() THEN
	RETURN;
END_IF

CASE _iState OF
START_DEVICE: 
	IF initDevice() < 0 THEN;
		goError(ReadWrite := FALSE);
		RETURN;	
	END_IF
	_iState := RUN_DEVICE;	
	mySteps := STEP_START_DEVICE;
	
RUN_DEVICE:
	CASE mySteps OF
		//Step for start device in cycle
		
		STEP_START_DEVICE:
		
			writeRequest.request := TRUE;
			IF NOT checkWriteTimeMultiplex(ADR(writeRequest)) THEN
				RETURN;
			END_IF
			IF setCommandRegister() < 0 THEN
				RETURN;
			END_IF
			IF startDevice() < 0 THEN
				RETURN;
			END_IF
			mySteps := STEP_READ;	
	END_CASE

	 
END_CASE
END_METHOD

METHOD initDevice : INT
VAR_INPUT
END_VAR
//set gain, integration time
//set gain, integration time depending on light intensity  
(*IF checkWrite8(TSL2561_TIMING_REGISTER_ADRESS OR TSL2561_COMMAND_REGISTER_BIT, (SHL(gain,4)OR integrationTime)) < 0 THEN
	RETURN;		
END_IF*)
//start device	
IF startDevice() < 0 THEN
	initDevice := ERROR_RET_VAL;
	RETURN;
END_IF

initDevice := WRITE_SUCCSESSFULL;
END_METHOD

METHOD checkDevice : bool
VAR_INPUT
END_VAR

VAR
	sensorData: ARRAY[0..0]OF BYTE;
END_VAR
checkDevice := FALSE;
IF checkReadRegister(TSL2561_ID_REGISTER_ADRESS OR TSL2561_BLOCK_COMMAND OR TSL2561_COMMAND_REGISTER_BIT, ADR(sensorData),1) < 0 THEN
	RETURN;
END_IF
IF (sensorData[0] AND 16#F0) <> 16#10 THEN
	//didn't found right sensor
	goError(ReadWrite := TRUE);
	RETURN;
END_IF	
checkDevice := TRUE;
END_METHOD

METHOD writeControlRegister : int
VAR_INPUT
END_VAR
END_METHOD

METHOD setCommandRegister:INT
VAR_INPUT
END_VAR
setCommandRegister := checkWrite8(TSL2561_TIMING_REGISTER_ADRESS OR TSL2561_COMMAND_REGISTER_BIT, (SHL(gain,4)OR integrationTime));
END_METHOD

METHOD startDevice : int
VAR_INPUT
END_VAR
startDevice := checkWrite8(TSL2561_CONTROLL_REGISTER_ADRESS OR TSL2561_COMMAND_REGISTER_BIT, TSL2561_DEVICE_START);
//set time for wait for next integration
waitIntegration := TICKS.GetTick(xDummy:=TRUE) + TSL2561_INTEGATION_TIME[integrationTime];
END_METHOD

METHOD stopDevice : int
VAR_INPUT
END_VAR
stopDevice := checkWrite8(TSL2561_CONTROLL_REGISTER_ADRESS OR TSL2561_COMMAND_REGISTER_BIT, TSL2561_DEVICE_STOP);
END_METHOD

METHOD getData : int
VAR_INPUT
END_VAR
VAR
	sensorData:ARRAY[0..3]OF BYTE;

END_VAR
(*read all sensor Data*)
getData := checkReadRegister(TSL2561_SENSOR_REGISTER_ADRESS OR TSL2561_BLOCK_COMMAND OR TSL2561_COMMAND_REGISTER_BIT, ADR(sensorData),4); 

//split data
fullData := WORD_TO_UINT(sensorData[0] OR (BYTE_TO_UINT(sensorData[1])*256));
irData := WORD_TO_UINT(sensorData[2] OR (BYTE_TO_UINT(sensorData[3])*256));
END_METHOD

METHOD calculateLux : int
VAR_INPUT
END_VAR
VAR 
	ratio:LREAL;
	ambient:LREAL;
	ir:LREAL;
	
END_VAR
//https://github.com/kc-GitHub/Wettersensor/blob/master/Firmware-Src/Libraries/TSL2561/TSL2561.cpp
IF gain = TSL2561_GAIN_LOW THEN
	ambient := UDINT_TO_LREAL(fullData) * 16;
	ir := UDINT_TO_LREAL(irData) * 16;
ELSE
	ambient := UDINT_TO_LREAL(fullData);
	ir := UDINT_TO_LREAL(irData);
END_IF
IF ambient = 0 THEN
	lux := 0;
	RETURN;
END_IF
ir := ir / TSL2561_INTEGRATION_TIME_SCALE[integrationTime];
ambient := ambient / TSL2561_INTEGRATION_TIME_SCALE[integrationTime];
ratio := ir / ambient;
IF (ratio >= 0) AND (ratio <= scale1CheckHigh) THEN
		lux := (scale1Calc1 * ambient) - (scale1Calc2 * ambient * (EXPT(ratio, 1.4)));
ELSIF ratio <= scale2CheckHigh THEN
		lux := (scale2Calc1 * ambient) - (scale2Calc2 * IR);
ELSIF ratio <= scale3CheckHigh THEN
		lux := (scale3Calc1 * ambient) - (scale3Calc2 * IR);
ELSIF ratio <= scale4CheckHigh THEN
		lux := (scale4Calc1 * ambient) - (scale4Calc2 * IR);
ELSIF ratio > scale5CheckHigh THEN
		lux := 0;
END_IF





(*
	ambient := fullData;
	ir := irData;
        (*Converts the raw sensor values to the standard SI lux equivalent.
        Returns 0 if the sensor is saturated and the values are unreliable.
        *)
        // Make sure the sensor isn't saturated!
        IF integrationTime = TSL2561_INTEGRATIONTIME_13MS THEN
            clipThreshold := TSL2561_CLIPPING_13MS;
        ELSIF integrationTime = TSL2561_INTEGRATIONTIME_101MS THEN
            clipThreshold := TSL2561_CLIPPING_101MS;
        ELSE
            clipThreshold := TSL2561_CLIPPING_402MS;
		END_IF

        // Return 0 lux if the sensor is saturated
        IF ambient > clipThreshold OR ir > clipThreshold THEN
            RETURN;
		END_IF
        //Get the correct scale depending on the integration time
        IF integrationTime = TSL2561_INTEGRATIONTIME_13MS THEN
            chScale := TSL2561_LUX_CHSCALE_TINT0;
        ELSIF integrationTime = TSL2561_INTEGRATIONTIME_101MS THEN
            chScale := TSL2561_LUX_CHSCALE_TINT1;
        ELSE
            chScale := SHL (TSL2561_LUX_CHSCALE,1);
		END_IF
        // Scale for gain (1x or 16x)
        IF gain = TSL2561_GAIN_HIGH THEN
            chScale := SHL(chScale,4);
		END_IF
        // Scale the channel values
        channel0 := SHR(ambient * chScale, TSL2561_LUX_CHSCALE);
        channel1 := SHR(ir * chScale, TSL2561_LUX_CHSCALE);

        // Find the ratio of the channel values (Channel1/Channel0)
        ratio1 := 0;
        IF channel0 <> 0 THEN
            ratio1 := SHL(channel1,TSL2561_LUX_RATIOSCALE + 1) / channel0;
		END_IF
        //round the ratio value
        ratio := SHR(ratio1 + 1, 1);

        b := 0;
        m := 0;

        IF ratio >= 0 AND ratio <= TSL2561_LUX_K1T THEN
            b := TSL2561_LUX_B1T;
            m := TSL2561_LUX_M1T;
        ELSIF ratio <= TSL2561_LUX_K2T THEN
            b := TSL2561_LUX_B2T;
            m := TSL2561_LUX_M2T;
        ELSIF ratio <= TSL2561_LUX_K3T THEN
            b := TSL2561_LUX_B3T;
            m := TSL2561_LUX_M3T;
        ELSIF ratio <= TSL2561_LUX_K4T THEN
            b := TSL2561_LUX_B4T;
            m := TSL2561_LUX_M4T;
        ELSIF ratio <= TSL2561_LUX_K5T THEN
            b := TSL2561_LUX_B5T;
            m := TSL2561_LUX_M5T;
        ELSIF ratio <= TSL2561_LUX_K6T THEN
            b := TSL2561_LUX_B6T;
            m := TSL2561_LUX_M6T;
        ELSIF ratio <= TSL2561_LUX_K7T THEN
            b := TSL2561_LUX_B7T;
            m := TSL2561_LUX_M7T;
        ELSIF ratio > TSL2561_LUX_K8T THEN
            b := TSL2561_LUX_B8T;
            m := TSL2561_LUX_M8T;
		END_IF
        temp := (channel0 * b) - (channel1 * m);

        //Do not allow negative lux value
        IF temp < 0 THEN
            temp := 0;
		END_IF

        //Round lsb (2^(LUX_SCALE-1))
        temp := temp +  SHL(1, TSL2561_LUX_LUXSCALE - 1);

        //Strip off fractional portion
        lux := SHR(temp, TSL2561_LUX_LUXSCALE);
*)
END_METHOD

END_FUNCTION_BLOCK

// Function Blocks/PCF8575IN
FUNCTION_BLOCK PCF8575IN EXTENDS I2C_BASE

VAR_OUTPUT
	ins: ARRAY[0..1] OF BYTE;
END_VAR

SUPER^();

METHOD Initialize : UDINT
VAR_INPUT
	wModuleType : UINT;
	dwInstance : UDINT;
	pConnector : POINTER TO IoConfigConnector;
END_VAR
VAR

END_VAR
SUPER^.Initialize(wModuleType, dwInstance, pConnector);


stateAfterError := RUN_DEVICE;
stateAfterInit := RUN_DEVICE;
END_METHOD

METHOD AfterReadInputs : INT
VAR

tmp : ARRAY[0..1] OF BYTE;

END_VAR
SUPER^.AfterReadInputs();

IF checkInitMultiplex() THEN
	RETURN;
END_IF

CASE _iState OF

RUN_DEVICE:
	//check if time are over
	IF NOT checkReadTimeMultiplex(ADR(readRequest)) THEN
		RETURN;
	END_IF
	IF checkRead(ADR(tmp),2) = READ_SUCCSESSFULL THEN
		ins := tmp;
	END_IF
	
END_CASE
END_METHOD

END_FUNCTION_BLOCK

// Function Blocks/PCA9685
{warning disable C0351}
{attribute 'setPWMRange'}
FUNCTION_BLOCK PCA9685 EXTENDS I2C_BASE
VAR_INPUT
	alrPWM: ARRAY[0..15] OF LREAL; 						(* 0..1 = 1ms..2ms Signal On *)
	alrBits: ARRAY[0..1]OF BYTE;
	axEnable: ARRAY[0..15] OF BOOL := [16(TRUE)];		(* Bit x = TRUE: set PWM output channel x; FALSE: do not modify output signal of channel x *)
END_VAR
VAR_OUTPUT
END_VAR
VAR
	_freq: UINT := 50;				(* frequency [Hz] *)

	_rPeriod: LREAL := 1.0;				(* Period [ms], time between two rising edges *)
	_alrOldPWM: ARRAY[0..15] OF UINT;
	_alrOldOnOff: ARRAY[0..1] OF BYTE;
	_alrPWM: ARRAY[0..15] OF UINT; //values for output
	_mode2:BYTE;
	_onOffMode: BOOL;

END_VAR
VAR_TEMP	
	i, usi: USINT;
END_VAR
{warning restore C0351}

SUPER^();

CASE _iState OF

START_INIT:
	writeRequest.request := TRUE;
	IF NOT checkWriteTimeMultiplex(ADR(writeRequest)) THEN
		RETURN;
	END_IF 
  	checkWrite8(GVL.PCA9685_MODE1, 16#10); // go to sleep

	usi := LREAL_TO_USINT(25000000 / 4096.0 / 0.88 (*0.88 after check with oszi*)  / _freq) - 1;
  	checkWrite8(GVL.PCA9685_PRESCALE, usi); // set the prescaler

	_rPeriod := LREAL#1.0 / _freq * 1000; //Periode in ms
	
  	_iState := START_DEVICE;
START_DEVICE:
	writeRequest.request := TRUE;
	IF NOT checkWriteTimeMultiplex(ADR(writeRequest)) THEN
		RETURN;
	END_IF
	 
  	checkWrite8(GVL.PCA9685_MODE1, 2#100000);  //  This sets the MODE1 register to turn on auto increment.
	checkWrite8(GVL.PCA9685_MODE2, _mode2);
	
	//force first write
	IF NOT _onOffMode THEN
		FOR i := 0 TO 15 DO
			_alrOldPWM[i] := 65000;
		END_FOR
	ELSE
		_alrOldOnOff[0] := NOT alrBits[0];
		_alrOldOnOff[1] := NOT alrBits[1];
	END_IF
	_iState := RUN_DEVICE;
END_CASE

METHOD BeforeWriteOutputs : INT
VAR
	aby: ARRAY[0..4] OF BYTE;
	i: USINT;
	tByte:BYTE;
	tByteIn:BYTE;
END_VAR
SUPER^.BeforeWriteOutputs();

IF checkInitMultiplex() THEN
	RETURN;
END_IF
IF _iState = RUN_DEVICE THEN
	IF _onOffMode THEN
		IF alrBits[0] <> _alrOldOnOff[0] THEN
			//Input did changed....
				tByte := alrBits[0] XOR _alrOldOnOff[0];
				tByteIn := alrBits[0];
			FOR i := 0 TO 7 DO
				IF tByte.0 THEN
					aby[0] := GVL.LED0_ON_L + 4 * i;
					IF tByteIn.0 THEN
						//set on
						aby[2].4 := FALSE;
						aby[4].4 := TRUE;  
						
					ELSE
						//set off
						aby[2].4 := TRUE;
						aby[4].4 := FALSE;  
						
					END_IF
					checkWrite(ADR(aby), 5);
				END_IF
				//shift one right
				tbyte := SHR(tbyte, 1);
				tByteIn := SHR(tbyteIn, 1);
			END_FOR
		END_IF
		IF alrBits[1] <> _alrOldOnOff[1] THEN
			 //Input did changed....
				tByte := alrBits[1] XOR _alrOldOnOff[1];
				tByteIn := alrBits[1];
			FOR i := 8 TO 15 DO
				IF tByte.0 THEN
					aby[0] := GVL.LED0_ON_L + 4 * i;
					IF tByteIn.0 THEN
						//set on
						aby[2].4 := FALSE;
						aby[4].4 := TRUE;  
						
					ELSE
						//set off
						aby[2].4 := TRUE;
						aby[4].4 := FALSE;  
						
					END_IF
					checkWrite(ADR(aby), 5);
				END_IF
				//shift one right
				tbyte := SHR(tbyte, 1);
				tByteIn := SHR(tbyteIn, 1);
			END_FOR
		END_IF
		//save new states
		_alrOldOnOff[0] := alrBits[0];
		_alrOldOnOff[1] := alrBits[1];
		
	ELSE
		IF calcOut() THEN
			writeRequest.request := TRUE;
		END_IF
		IF NOT checkWriteTimeMultiplex(ADR(writeRequest)) THEN
			RETURN;
		END_IF 
		FOR i:=0 TO 15 DO
			IF _alrPWM[i] <> _alrOldPWM[i] AND axEnable[i]  THEN
				_alrOldPWM[i] := _alrPWM[i];//slave new value
					
				aby[0] := GVL.LED0_ON_L + 4 * i;
				aby[3] := UINT_TO_USINT(_alrPWM[i]);
				aby[4] := UINT_TO_USINT(_alrPWM[i]/256);
	
				checkWrite(ADR(aby), 5);
	
			END_IF
		END_FOR	
	END_IF
END_IF
END_METHOD

METHOD Initialize : UDINT
VAR_INPUT
	wModuleType : UINT;
	dwInstance : UDINT;
	pConnector : POINTER TO IoConfigConnector;
END_VAR
VAR
	pParam: POINTER TO IoConfigParameter;		
	udiResult: UDINT;
END_VAR
SUPER^.Initialize(wModuleType, dwInstance, pConnector);

//get frequenzie
pParam := ConfigGetParameter(_pConnector, 20);
IF pParam <> 0 THEN
	_freq := IoStandard.ConfigGetParameterValueWord(pParam, ADR(udiResult));
END_IF

pParam := ConfigGetParameter(_pConnector, 21);
IF pParam <> 0 THEN
	_mode2 := IoStandard.ConfigGetParameterValueByte(pParam, ADR(udiResult));
END_IF
//get on/off Mode
_onOffMode := _mode2.5;
//delet it in control byte
_mode2.5 := FALSE; 

stateAfterError := START_DEVICE;
stateAfterInit := START_DEVICE;
END_METHOD

METHOD calcOut : bool
calcOut := FALSE;	
FOR i:=0 TO 15 DO
	IF  axEnable[i] > 0 THEN
		_alrPWM[i] := LREAL_TO_UINT(LIMIT(0, alrPWM[i], 1) * 4095);
		IF _alrPWM[i] <> _alrOldPWM[i] THEN
			calcOut := TRUE;
			
		END_IF
	END_IF
END_FOR
END_METHOD

END_FUNCTION_BLOCK

// Function Blocks/Dim4Ch
(*for 4 ch 230V Phase Dimmer from ebay, only runs under 100Hz!!!!*)

FUNCTION_BLOCK Dim4Ch EXTENDS I2C_BASE
VAR_INPUT
	alrDim: ARRAY[0..3] OF BYTE; 						(* 0..1 = 1ms..2ms Signal On *)
	axEnable: ARRAY[0..3] OF BOOL := [4(TRUE)];		(* Bit x = TRUE: set PWM output channel x; FALSE: do not modify output signal of channel x *)
	fastOut:BOOL;//try to output more than one channel if changed 
END_VAR
VAR_OUTPUT
END_VAR
VAR
	_alrOldDim: ARRAY[0..3] OF USINT;
	_alrDim: ARRAY[0..3] OF USINT; //values for output
END_VAR
VAR_TEMP	
	i, usi: USINT;
END_VAR
VAR CONSTANT
	channelAdress:ARRAY[0..3]OF BYTE :=[16#80,16#81,16#82,16#83];
END_VAR

SUPER^();


CASE _iState OF

START_DEVICE:
	IF usiAddress = 0 THEN
		usiAddress := 16#27;
	END_IF
	//force first write
	FOR i := 0 TO 3 DO
		_alrOldDim[i] := 101;
	END_FOR
	
	_iState := RUN_DEVICE;
END_CASE

METHOD BeforeWriteOutputs : INT
VAR
	aby: ARRAY[0..7] OF BYTE;
	i: USINT;
	channelCount:USINT;
END_VAR
SUPER^.BeforeWriteOutputs();

IF checkInitMultiplex() THEN
	RETURN;
END_IF

IF _iState = RUN_DEVICE THEN
	IF calcOut() THEN
		writeRequest.request := TRUE;
	END_IF
	IF (NOT isMultiplex AND NOT writeRequest.request) OR (NOT checkWriteTimeMultiplex(ADR(writeRequest)) AND isMultiplex) THEN
		RETURN;
	END_IF 
	writeRequest.request := FALSE;
	IF fastOut THEN
		channelCount := 0;
		FOR i:=0 TO 3 DO
			IF _alrDim[i] <> _alrOldDim[i] AND axEnable[i]  THEN
				_alrOldDim[i] := _alrDim[i];//slave new value
					
				aby[channelCount*2] := channelAdress[i];
				aby[channelCount*2+1] := UINT_TO_USINT(_alrDim[i]);
				channelCount := channelCount + 1;
	
			END_IF
		END_FOR
		checkWrite(ADR(aby), channelCount*2);
	ELSE
		FOR i:=0 TO 3 DO
			IF _alrDim[i] <> _alrOldDim[i] AND axEnable[i]  THEN
				_alrOldDim[i] := _alrDim[i];//slave new value
					
				aby[0] := channelAdress[i];
				aby[1] := _alrDim[i];
				checkWrite(ADR(aby), 2);
				//checkWrite(ADR(aby)+1, 1);
				//checkWrite8(channelAdress[i], _alrDim[i]);
	
			END_IF
		END_FOR	
	END_IF
END_IF
END_METHOD

METHOD Initialize : UDINT
VAR_INPUT
	wModuleType : UINT;
	dwInstance : UDINT;
	pConnector : POINTER TO IoConfigConnector;
END_VAR
VAR
	pParam: POINTER TO IoConfigParameter;		
	udiResult: UDINT;
END_VAR
SUPER^.Initialize(wModuleType, dwInstance, pConnector);


pParam := ConfigGetParameter(_pConnector, 1);
IF pParam <> 0 THEN	//store own pointer in this param
	pParam^.dwDriverSpecific := THIS;
END_IF

stateAfterError := START_DEVICE;
stateAfterInit := START_DEVICE;
END_METHOD

METHOD calcOut : bool
calcOut := FALSE;	
FOR i:=0 TO 3 DO
	IF  axEnable[i] > 0 THEN
		_alrDim[i] := 100 - LIMIT(0, alrDim[i],100);
		IF _alrDim[i] <> _alrOldDim[i] THEN
			calcOut := TRUE;
			
		END_IF
	END_IF
END_FOR
END_METHOD

END_FUNCTION_BLOCK

// Function Blocks/EEPROM_24C512
FUNCTION_BLOCK EEPROM_24C512 EXTENDS I2C_BASE
VAR_IN_OUT
	
END_VAR
VAR_INPUT
	DATA:POINTER TO CommonTypesAndFunctions.EEPROM_DATA;
END_VAR
VAR_OUTPUT
END_VAR
VAR
	pResult:SysSem.RTS_IEC_RESULT;
END_VAR

SUPER^();



IF DATA = 0 THEN RETURN; END_IF 




IF NOT DATA^.HANDLE_VALID THEN
	//get semaphore
	DATA^.SEMAPHORE := SysSemCreate(pResult:= ADR(pResult));
	DATA^.HANDLE_VALID := TRUE;
	DATA^.SIZE_OF_VALUE := SIZEOF(DATA^.VALUE_IN);
END_IF

METHOD Initialize : UDINT
VAR_INPUT
	wModuleType : UINT;
	dwInstance : UDINT;
	pConnector : POINTER TO IoConfigConnector;
END_VAR
VAR

END_VAR
SUPER^.Initialize(wModuleType, dwInstance, pConnector);


stateAfterError := RUN_DEVICE;
stateAfterInit := RUN_DEVICE;
END_METHOD

METHOD AfterReadInputs : INT
VAR

	pyBuffer:ARRAY[0..1] OF BYTE;
 	pResult:SysSem.RTS_IEC_RESULT;
END_VAR
SUPER^.AfterReadInputs();

IF DATA = 0 THEN RETURN; END_IF 

IF checkInitMultiplex() THEN
	RETURN;
END_IF

CASE _iState OF

RUN_DEVICE:

	IF SysSem.SysSemEnter(hSem:=DATA^.SEMAPHORE) = SysSem.Errors.ERR_OK THEN
	
		IF DATA^.FB_NO_IN > 0 THEN 
			//IF DATA := 0 THEN RETURN; END_IF//didnt get a pointer jet
			IF DATA^.READ_PAGE OR DATA^.READ_VALUE THEN
				readRequest.request := TRUE;
			END_IF
			
			//check if request is done
			IF checkReadTimeMultiplex(ADR(readRequest)) THEN
				readRequest.request := FALSE;
				IF DATA^.READ_PAGE THEN
					//first write Page adress
					pyBuffer[0]:=MEM.HighByte(wValue:= DATA^.ADDRESS_PAGE);
					pyBuffer[1]:=MEM.LowByte(wValue:= DATA^.ADDRESS_PAGE);
					
					IF checkWrite(ADR(pyBuffer), SIZEOF(pyBuffer)) = WRITE_SUCCSESSFULL THEN 
					//now read the page
					
						IF checkRead(ADR(DATA^.PAGE_OUT), SIZEOF(DATA^.PAGE_OUT)) = READ_SUCCSESSFULL THEN
							DATA^.READ_PAGE := FALSE;		
							DATA^.FB_NO_OUT := DATA^.FB_NO_IN;
							DATA^.FB_NO_IN := 0;
						END_IF;
					END_IF;
				END_IF
				
				IF DATA^.READ_VALUE THEN
					//first write VAR adress
					pyBuffer[0]:=MEM.HighByte(wValue:= DATA^.ADDRESS_VALUE);
					pyBuffer[1]:=MEM.LowByte(wValue:= DATA^.ADDRESS_VALUE);
					
					IF checkWrite(ADR(pyBuffer), SIZEOF(pyBuffer)) = WRITE_SUCCSESSFULL THEN 
					//now read the VAR
					
						IF checkRead(ADR(DATA^.VALUE_OUT), SIZEOF(DATA^.VALUE_OUT)) = READ_SUCCSESSFULL THEN 
							DATA^.READ_VALUE := FALSE;
							DATA^.FB_NO_OUT := DATA^.FB_NO_IN;
							DATA^.FB_NO_IN := 0;
						END_IF;
					END_IF;
				END_IF
			END_IF
		END_IF
	SysSem.SysSemLeave(hSem:=DATA^.SEMAPHORE);	
	END_IF	
END_CASE
END_METHOD

METHOD BeforeWriteOutputs : INT
VAR
 pyBuffer:ARRAY[0..128-1+2] OF BYTE;
 PART_HIGH:UINT;
 SIZE_OF_ADDRESS:UINT;
 pResult:SysSem.RTS_IEC_RESULT;
END_VAR
SUPER^.BeforeWriteOutputs();

IF DATA = 0 THEN RETURN; END_IF

IF checkInitMultiplex() THEN
	RETURN;
END_IF


CASE _iState OF


RUN_DEVICE:
	IF SysSem.SysSemEnter(hSem:=DATA^.SEMAPHORE) = SysSem.Errors.ERR_OK THEN
	
			//requestWrite
			IF DATA^.WRITE_PAGE OR DATA^.WRITE_VALUE THEN
				writeRequest.request := TRUE;
			END_IF
			//check if request is done
			IF checkWriteTimeMultiplex(ADR(writeRequest)) THEN
				
			
				//reset request
				writeRequest.request := FALSE;	
				
				IF DATA^.WRITE_PAGE THEN
					
					//checkWrite(ADR(pyBuffer),3);
					MEM.MemMove(pSource:= ADR(DATA^.PAGE_IN), pDestination:= ADR(pyBuffer[2]), uiNumberOfBytes:= DATA^.PAGE_SIZE);
					//Addresse in Puffer dazu...
					pyBuffer[0]:=MEM.HighByte(wValue:= DATA^.ADDRESS_PAGE);
					pyBuffer[1]:=MEM.LowByte(wValue:= DATA^.ADDRESS_PAGE AND 2#10000000);
				
					IF checkWrite(ADR(pyBuffer),SIZEOF(pyBuffer)) = WRITE_SUCCSESSFULL THEN 
					
						DATA^.WRITE_PAGE := FALSE;
						DATA^.FB_NO_IN := 0;//reset request
					END_IF;
				END_IF
				
				IF DATA^.WRITE_VALUE THEN
					//here we have the Problem of the page Write, if we swap over an page border by writing values
					//we jump to byte 0 of current page and an different address... so write every byte one by one,
					//or check borders...
					
					//so, lets chek borders
					
					SIZE_OF_ADDRESS := 2;
					
					IF DATA^.ADDRESS_VALUE MOD DATA^.PAGE_SIZE + SIZEOF(CommonTypesAndFunctions.ALL_TYPES_UNION) > DATA^.PAGE_SIZE THEN
						PART_HIGH := DATA^.PAGE_SIZE - DATA^.ADDRESS_VALUE MOD DATA^.PAGE_SIZE;
						MEM.MemMove(pSource:= ADR(DATA^.VALUE_IN), pDestination:= ADR(pyBuffer[2]),
									 uiNumberOfBytes:= PART_HIGH);
						pyBuffer[0]:=MEM.HighByte(wValue:= DATA^.ADDRESS_VALUE);
						pyBuffer[1]:=MEM.LowByte(wValue:= DATA^.ADDRESS_VALUE);
						//write first part
						IF checkWrite(ADR(pyBuffer),PART_HIGH + SIZE_OF_ADDRESS) = WRITE_SUCCSESSFULL THEN 
							//write second part
							pyBuffer[0]:=MEM.HighByte(wValue:= DATA^.ADDRESS_VALUE + PART_HIGH);
							pyBuffer[1]:=MEM.LowByte(wValue:= DATA^.ADDRESS_VALUE + PART_HIGH);
							MEM.MemMove(pSource:= ADR(DATA^.VALUE_IN) + PART_HIGH, pDestination:= ADR(pyBuffer[2]),
										 uiNumberOfBytes:= SIZEOF(CommonTypesAndFunctions.ALL_TYPES_UNION)  - PART_HIGH);
							IF checkWrite(ADR(pyBuffer),SIZEOF(CommonTypesAndFunctions.ALL_TYPES_UNION)  - PART_HIGH + SIZE_OF_ADDRESS) = WRITE_SUCCSESSFULL THEN
 								DATA^.WRITE_VALUE := FALSE;
								DATA^.FB_NO_IN := 0;//reset request
							END_IF;
						END_IF;
					ELSE//here i can write without thinking about pages
						MEM.MemMove(pSource:= ADR(DATA^.VALUE_IN), pDestination:= ADR(pyBuffer[2]), uiNumberOfBytes:= SIZEOF(CommonTypesAndFunctions.EEPROM_DATA));
						pyBuffer[0]:=MEM.HighByte(wValue:= DATA^.ADDRESS_VALUE);
						pyBuffer[1]:=MEM.LowByte(wValue:= DATA^.ADDRESS_VALUE);
						IF checkWrite(ADR(pyBuffer),SIZEOF(CommonTypesAndFunctions.ALL_TYPES_UNION)+ SIZE_OF_ADDRESS) = WRITE_SUCCSESSFULL THEN 
							DATA^.WRITE_VALUE := FALSE;
							DATA^.FB_NO_IN := 0;//reset request
						
						END_IF;
					END_IF
				END_IF
			END_IF
	SysSem.SysSemLeave(hSem:=DATA^.SEMAPHORE);	
	END_IF		
END_CASE
END_METHOD

END_FUNCTION_BLOCK

// Function Blocks/SSD1306
FUNCTION_BLOCK SSD1306 EXTENDS I2C_BASE


(*

bit order:
byte:	  0 1 2 3 4 5 6 7 8 9 10
	 	 _ _ _ _ _ _ _ _ _ _ _ _ _ _ _ _
bit:	0|_|_|_|_|_|_|_|_|_|_|_|_|_|_|_|_|
		1|_|_|_|_|_|_|_|_|_|_|_|_|_|_|_|_|
		2|_|_|_|_|_|_|_|_|_|_|_|_|_|_|_|_|
		3|_|_|_|_|_|_|_|_|_|_|_|_|_|_|_|_|
		4|_|_|_|_|_|_|_|_|_|_|_|_|_|_|_|_|
		5|_|_|_|_|_|_|_|_|_|_|_|_|_|_|_|_|
		6|_|_|_|_|_|_|_|_|_|_|_|_|_|_|_|_|
		7|_|_|_|_|_|_|_|_|_|_|_|_|_|_|_|_|
		0|_|_|_|_|_|_|_|_|_|_|_|_|_|_|_|_|
		1|_|_|_|_|_|_|_|_|_|_|_|_|_|_|_|_|
		2|_|_|_|_|_|_|_|_|_|_|_|_|_|_|_|_|
cursor:
X:=0; Y:= 0 = upper left corner, alsoght for soft font
Fonts from:
https://github.com/basti79/LCD-fonts
http://en.pudn.com/downloads180/sourcecode/embed/detail838497_en.html
MSB 1 vertikal
*)
VAR_INPUT
	
	
END_VAR
VAR



	displayHeight:USINT;
	displayWidth:USINT;
	displaySize:USINT;
	
	displayBuffer:ARRAY[0..1024]OF BYTE := [16#40];//one Byte more fore Command Byte
	//displayBuffer:ARRAY[0..1024]OF BYTE := [16#40, 1024(2#1)];//one Byte more fore Command Byte
	
	writeRequestLCDData: BOOL;
	writeRequestLCDCommand: BOOL;
	displayOnOff: BOOL;

	bytesPerRow:UINT;
	pixPerByte:USINT := 8;
	
	commandBuffer:ARRAY[0..9] OF BYTE:= [16#00];//Buffer for commands
	sizeOfCommands:USINT := 1;
	lastBufferWriteTime:CAA.TICK;
	
	(**************************************************************************************************************)
	
	//VARs for SoftFont
	aktFont:USINT;

	cursorX:USINT;
	cursorY:USINT;
	cursorBaseX:USINT;
	cursorBaseY:USINT;
		
	
	(**************************************************************************************************************)
	//start sequens
	initDisplayData: ARRAY[0..27]OF BYTE :=[16#00,//Command code
	16#AE,			// Display OFF (sleep mode)
	16#20, 16#00,		// Set Memory Addressing Mode
					// 00=Horizontal Addressing Mode; 01=Vertical Addressing Mode;
					// 10=Page Addressing Mode (RESET); 11=Invalid
	16#B0,			// Set Page Start Address for Page Addressing Mode, 0-7
	16#C8,			// Set COM Output Scan Direction
	16#00,			// --set low column address
	16#10,			// --set high column address
	16#40,			// --set start line address
	16#81, 16#3F,		// Set contrast control register
	16#A1,			// Set Segment Re-map. A0=address mapped; A1=address 127 mapped.
	16#A6,			// Set display mode. A6=Normal; A7=Inverse
	
	16#A4,			// Output RAM to Display
					// 16#A4=Output follows RAM content; 16#A5,Output ignores RAM content
	16#D3, 16#00,		// Set display offset. 00 = no offset
	16#D5,			// --set display clock divide ratio/oscillator frequency
	16#F0,			// --set divide ratio
	16#D9, 16#22,		// Set pre-charge period
	16#DA, 16#12,		// Set com pins hardware configuration		
	16#DB,			// --set vcomh
	16#20,			// 16#20,0.77xVcc
	16#8D, 16#14		// Set DC-DC enable
//	16#AF			// Display ON
	];

	
END_VAR

VAR CONSTANT 
	
//bitMask:ARRAY[0..7]OF BYTE :=[128, 64, 32, 16, 8, 4, 2, 1];
bitMask:ARRAY[0..7]OF BYTE :=[1, 2, 4, 8, 16, 32, 64, 128];
//FONT_16X26
softFontData:ARRAY[0..14] OF SOFT_FONT_DATA := [(width:=4, height:=6, mask:=2#11_111100, data:=ADR(FONT_4X6), size:=4),
												(width:=5, height:=8, mask:=2#1111_1111, data:=ADR(FONT_5X8), size:=5),
												(width:=5, height:=12, mask:=2#1111_1111_1111_0000, data:=ADR(FONT_5X12), size:=10),
												(width:=6, height:=8, mask:=2#1111_1111, data:=ADR(FONT_6X8), size:=6),
												(width:=6, height:=10, mask:=2#1111_1111_1100_0000, data:=ADR(FONT_6X10), size:=12),
												(width:=7, height:=12, mask:=2#1111_1111_1111_0000, data:=ADR(FONT_7X12), size:=14),
												(width:=7, height:=12, mask:=2#1111_1111_1111_0000, data:=ADR(FONT_7X12B), size:=14),
												(width:=8, height:=8, mask:=2#1111_1111, data:=ADR(FONT_8X8), size:=8),
												(width:=8, height:=12, mask:=2#1111_1111_1111_0000, data:=ADR(FONT_8X12), size:=16),
												(width:=8, height:=14, mask:=2#1111_1111_1111_1100, data:=ADR(FONT_8X14), size:=16),
												(width:=10, height:=16, mask:=2#1111_1111_1111_1111, data:=ADR(FONT_10X16), size:=20),
												(width:=12, height:=16, mask:=2#1111_1111_1111_1111, data:=ADR(FONT_12X16), size:=24),
												(width:=16, height:=8, mask:=2#1111_1111, data:=ADR(FONT_16X8), size:=16),
												(width:=16, height:=12, mask:=2#1111_1111_1111_0000, data:=ADR(FONT_16X12), size:=32),
												(width:=16, height:=26, mask:=2#11_1111_1111_1111_1111_1111_1111_0000, data:=ADR(FONT_16X26), size:=52)];


byteMask:ARRAY[0..15]OF BYTE := [2#11111111,
								2#01111111,
								2#00111111,
								2#00011111,
								2#00001111,
								2#00000111,
								2#00000011,
								2#00000001,
								
								2#10000000,
								2#11000000,
								2#11100000,
								2#11110000,
								2#11111000,
								2#11111100,
								2#11111110,
								2#11111111];


ssd1306oled_font6x8:ARRAY[0..5000]OF BYTE := [
    16#00, 16#00, 16#00, 16#00, 16#00, 16#00, // sp
    16#00, 16#00, 16#00, 16#2f, 16#00, 16#00, // !
    16#00, 16#00, 16#07, 16#00, 16#07, 16#00, // "
    16#00, 16#14, 16#7f, 16#14, 16#7f, 16#14, // #
    16#00, 16#24, 16#2a, 16#7f, 16#2a, 16#12, // $
    16#00, 16#62, 16#64, 16#08, 16#13, 16#23, // %
    16#00, 16#36, 16#49, 16#55, 16#22, 16#50, // &
    16#00, 16#00, 16#05, 16#03, 16#00, 16#00, // '
    16#00, 16#00, 16#1c, 16#22, 16#41, 16#00, // (
    16#00, 16#00, 16#41, 16#22, 16#1c, 16#00, // )
    16#00, 16#14, 16#08, 16#3E, 16#08, 16#14, // *
    16#00, 16#08, 16#08, 16#3E, 16#08, 16#08, // +
    16#00, 16#00, 16#00, 16#A0, 16#60, 16#00, // ,
    16#00, 16#08, 16#08, 16#08, 16#08, 16#08, // -
    16#00, 16#00, 16#60, 16#60, 16#00, 16#00, // .
    16#00, 16#20, 16#10, 16#08, 16#04, 16#02, // /
    16#00, 16#3E, 16#51, 16#49, 16#45, 16#3E, // 0
    16#00, 16#00, 16#42, 16#7F, 16#40, 16#00, // 1
    16#00, 16#42, 16#61, 16#51, 16#49, 16#46, // 2
    16#00, 16#21, 16#41, 16#45, 16#4B, 16#31, // 3
    16#00, 16#18, 16#14, 16#12, 16#7F, 16#10, // 4
    16#00, 16#27, 16#45, 16#45, 16#45, 16#39, // 5
    16#00, 16#3C, 16#4A, 16#49, 16#49, 16#30, // 6
    16#00, 16#01, 16#71, 16#09, 16#05, 16#03, // 7
    16#00, 16#36, 16#49, 16#49, 16#49, 16#36, // 8
    16#00, 16#06, 16#49, 16#49, 16#29, 16#1E, // 9
    16#00, 16#00, 16#36, 16#36, 16#00, 16#00, // :
    16#00, 16#00, 16#56, 16#36, 16#00, 16#00, // ;
    16#00, 16#08, 16#14, 16#22, 16#41, 16#00, // <
    16#00, 16#14, 16#14, 16#14, 16#14, 16#14, // =
    16#00, 16#00, 16#41, 16#22, 16#14, 16#08, // >
    16#00, 16#02, 16#01, 16#51, 16#09, 16#06, // ?
    16#00, 16#32, 16#49, 16#59, 16#51, 16#3E, // @
    16#00, 16#7C, 16#12, 16#11, 16#12, 16#7C, // A
    16#00, 16#7F, 16#49, 16#49, 16#49, 16#36, // B
    16#00, 16#3E, 16#41, 16#41, 16#41, 16#22, // C
    16#00, 16#7F, 16#41, 16#41, 16#22, 16#1C, // D
    16#00, 16#7F, 16#49, 16#49, 16#49, 16#41, // E
    16#00, 16#7F, 16#09, 16#09, 16#09, 16#01, // F
    16#00, 16#3E, 16#41, 16#49, 16#49, 16#7A, // G
    16#00, 16#7F, 16#08, 16#08, 16#08, 16#7F, // H
    16#00, 16#00, 16#41, 16#7F, 16#41, 16#00, // I
    16#00, 16#20, 16#40, 16#41, 16#3F, 16#01, // J
    16#00, 16#7F, 16#08, 16#14, 16#22, 16#41, // K
    16#00, 16#7F, 16#40, 16#40, 16#40, 16#40, // L
    16#00, 16#7F, 16#02, 16#0C, 16#02, 16#7F, // M
    16#00, 16#7F, 16#04, 16#08, 16#10, 16#7F, // N
    16#00, 16#3E, 16#41, 16#41, 16#41, 16#3E, // O
    16#00, 16#7F, 16#09, 16#09, 16#09, 16#06, // P
    16#00, 16#3E, 16#41, 16#51, 16#21, 16#5E, // Q
    16#00, 16#7F, 16#09, 16#19, 16#29, 16#46, // R
    16#00, 16#46, 16#49, 16#49, 16#49, 16#31, // S
    16#00, 16#01, 16#01, 16#7F, 16#01, 16#01, // T
    16#00, 16#3F, 16#40, 16#40, 16#40, 16#3F, // U
    16#00, 16#1F, 16#20, 16#40, 16#20, 16#1F, // V
    16#00, 16#3F, 16#40, 16#38, 16#40, 16#3F, // W
    16#00, 16#63, 16#14, 16#08, 16#14, 16#63, // X
    16#00, 16#07, 16#08, 16#70, 16#08, 16#07, // Y
    16#00, 16#61, 16#51, 16#49, 16#45, 16#43, // Z
    16#00, 16#00, 16#7F, 16#41, 16#41, 16#00, // [
    16#00, 16#55, 16#2A, 16#55, 16#2A, 16#55, // backslash
    16#00, 16#00, 16#41, 16#41, 16#7F, 16#00, // ]
    16#00, 16#04, 16#02, 16#01, 16#02, 16#04, // ^
    16#00, 16#40, 16#40, 16#40, 16#40, 16#40, // _
    16#00, 16#00, 16#01, 16#02, 16#04, 16#00, // '
    16#00, 16#20, 16#54, 16#54, 16#54, 16#78, // a
    16#00, 16#7F, 16#48, 16#44, 16#44, 16#38, // b
    16#00, 16#38, 16#44, 16#44, 16#44, 16#20, // c
    16#00, 16#38, 16#44, 16#44, 16#48, 16#7F, // d
    16#00, 16#38, 16#54, 16#54, 16#54, 16#18, // e
    16#00, 16#08, 16#7E, 16#09, 16#01, 16#02, // f
    16#00, 16#18, 16#A4, 16#A4, 16#A4, 16#7C, // g
    16#00, 16#7F, 16#08, 16#04, 16#04, 16#78, // h
    16#00, 16#00, 16#44, 16#7D, 16#40, 16#00, // i
    16#00, 16#40, 16#80, 16#84, 16#7D, 16#00, // j
    16#00, 16#7F, 16#10, 16#28, 16#44, 16#00, // k
    16#00, 16#00, 16#41, 16#7F, 16#40, 16#00, // l
    16#00, 16#7C, 16#04, 16#18, 16#04, 16#78, // m
    16#00, 16#7C, 16#08, 16#04, 16#04, 16#78, // n
    16#00, 16#38, 16#44, 16#44, 16#44, 16#38, // o
    16#00, 16#FC, 16#24, 16#24, 16#24, 16#18, // p
    16#00, 16#18, 16#24, 16#24, 16#18, 16#FC, // q
    16#00, 16#7C, 16#08, 16#04, 16#04, 16#08, // r
    16#00, 16#48, 16#54, 16#54, 16#54, 16#20, // s
    16#00, 16#04, 16#3F, 16#44, 16#40, 16#20, // t
    16#00, 16#3C, 16#40, 16#40, 16#20, 16#7C, // u
    16#00, 16#1C, 16#20, 16#40, 16#20, 16#1C, // v
    16#00, 16#3C, 16#40, 16#30, 16#40, 16#3C, // w
    16#00, 16#44, 16#28, 16#10, 16#28, 16#44, // x
    16#00, 16#1C, 16#A0, 16#A0, 16#A0, 16#7C, // y
    16#00, 16#44, 16#64, 16#54, 16#4C, 16#44, // z
	16#00, 16#00, 16#08, 16#77, 16#41, 16#00, // {
	16#00, 16#00, 16#00, 16#63, 16#00, 16#00, // ¦
	16#00, 16#00, 16#41, 16#77, 16#08, 16#00, // }
	16#00, 16#08, 16#04, 16#08, 16#08, 16#04, // ~
	16#00, 16#3D, 16#40, 16#40, 16#20, 16#7D, // ü
	16#00, 16#3D, 16#40, 16#40, 16#40, 16#3D, // Ü
	16#00, 16#21, 16#54, 16#54, 16#54, 16#79, // ä
	16#00, 16#7D, 16#12, 16#11, 16#12, 16#7D, // Ä
	16#00, 16#39, 16#44, 16#44, 16#44, 16#39, // ö
	16#00, 16#3D, 16#42, 16#42, 16#42, 16#3D, // Ö
	16#00, 16#02, 16#05, 16#02, 16#00, 16#00, // °
	16#00, 16#7E, 16#01, 16#49, 16#55, 16#73 // ß
];


FONT_4X6: ARRAY[0..255,0..3] OF BYTE :=[
16#00,16#00,16#00,16#00,	// 16#00
16#00,16#0E,16#15,16#0E,	// 16#01
16#00,16#0E,16#1B,16#0E,	// 16#02
16#00,16#0E,16#1C,16#0E,	// 16#03
16#00,16#0C,16#1E,16#0C,	// 16#04
16#00,16#16,16#1F,16#16,	// 16#05
16#00,16#14,16#1F,16#14,	// 16#06
16#00,16#00,16#00,16#00,	// 16#07
16#00,16#00,16#00,16#00,	// 16#08
16#00,16#00,16#00,16#00,	// 16#09
16#00,16#00,16#00,16#00,	// 16#0A
16#00,16#18,16#1A,16#06,	// 16#0B
16#00,16#0A,16#1D,16#0A,	// 16#0C
16#00,16#00,16#00,16#00,	// 16#0D
16#00,16#04,16#13,16#0E,	// 16#0E
16#00,16#0E,16#1B,16#0E,	// 16#0F
16#00,16#1F,16#0E,16#04,	// 16#10
16#00,16#04,16#0E,16#1F,	// 16#11
16#00,16#0A,16#1F,16#0A,	// 16#12
16#00,16#17,16#00,16#17,	// 16#13
16#00,16#00,16#3C,16#02,	// 16#14
16#00,16#10,16#0F,16#00,	// 16#15
16#00,16#10,16#10,16#10,	// 16#16
16#00,16#2A,16#3F,16#2A,	// 16#17
16#00,16#02,16#1F,16#02,	// 16#18
16#00,16#08,16#1F,16#08,	// 16#19
16#04,16#04,16#0E,16#04,	// 16#1A
16#04,16#0E,16#04,16#04,	// 16#1B
16#00,16#0C,16#08,16#08,	// 16#1C
16#00,16#0E,16#04,16#0E,	// 16#1D
16#00,16#0C,16#0E,16#0C,	// 16#1E
16#00,16#06,16#0E,16#06,	// 16#1F
16#00,16#00,16#00,16#00,	// 16#20
16#00,16#00,16#17,16#00,	// 16#21
16#00,16#03,16#00,16#03,	// 16#22
16#00,16#1F,16#0A,16#1F,	// 16#23
16#00,16#14,16#3F,16#0A,	// 16#24
16#00,16#09,16#04,16#12,	// 16#25
16#00,16#1A,16#15,16#1E,	// 16#26
16#00,16#03,16#01,16#00,	// 16#27
16#00,16#0E,16#11,16#00,	// 16#28
16#00,16#11,16#0E,16#00,	// 16#29
16#00,16#15,16#0E,16#15,	// 16#2A
16#00,16#04,16#0E,16#04,	// 16#2B
16#00,16#30,16#10,16#00,	// 16#2C
16#00,16#04,16#04,16#04,	// 16#2D
16#00,16#00,16#10,16#00,	// 16#2E
16#00,16#18,16#04,16#03,	// 16#2F
16#00,16#1E,16#11,16#0F,	// 16#30
16#00,16#12,16#1F,16#10,	// 16#31
16#00,16#19,16#15,16#12,	// 16#32
16#00,16#11,16#15,16#0A,	// 16#33
16#00,16#06,16#04,16#1F,	// 16#34
16#00,16#17,16#15,16#09,	// 16#35
16#00,16#0E,16#15,16#08,	// 16#36
16#00,16#01,16#1D,16#07,	// 16#37
16#00,16#0A,16#15,16#0A,	// 16#38
16#00,16#02,16#15,16#0E,	// 16#39
16#00,16#00,16#14,16#00,	// 16#3A
16#00,16#30,16#14,16#00,	// 16#3B
16#00,16#04,16#0A,16#11,	// 16#3C
16#00,16#14,16#14,16#14,	// 16#3D
16#00,16#11,16#0A,16#04,	// 16#3E
16#00,16#01,16#15,16#02,	// 16#3F
16#00,16#1F,16#11,16#17,	// 16#40
16#00,16#1E,16#05,16#1E,	// 16#41
16#00,16#1F,16#15,16#0A,	// 16#42
16#00,16#0E,16#11,16#11,	// 16#43
16#00,16#1F,16#11,16#0E,	// 16#44
16#00,16#1F,16#15,16#11,	// 16#45
16#00,16#1F,16#05,16#01,	// 16#46
16#00,16#0E,16#11,16#1D,	// 16#47
16#00,16#1F,16#04,16#1F,	// 16#48
16#00,16#11,16#1F,16#11,	// 16#49
16#00,16#08,16#10,16#0F,	// 16#4A
16#00,16#1F,16#04,16#1B,	// 16#4B
16#00,16#1F,16#10,16#10,	// 16#4C
16#00,16#1F,16#06,16#1F,	// 16#4D
16#00,16#1F,16#02,16#1F,	// 16#4E
16#00,16#0E,16#11,16#0E,	// 16#4F
16#00,16#1F,16#05,16#02,	// 16#50
16#00,16#0E,16#19,16#1E,	// 16#51
16#00,16#1F,16#05,16#1A,	// 16#52
16#00,16#16,16#15,16#0D,	// 16#53
16#00,16#01,16#1F,16#01,	// 16#54
16#00,16#1F,16#10,16#1F,	// 16#55
16#00,16#0F,16#10,16#0F,	// 16#56
16#00,16#1F,16#0C,16#1F,	// 16#57
16#00,16#1B,16#04,16#1B,	// 16#58
16#00,16#03,16#1C,16#03,	// 16#59
16#00,16#19,16#15,16#13,	// 16#5A
16#00,16#1F,16#11,16#00,	// 16#5B
16#00,16#03,16#04,16#18,	// 16#5C
16#00,16#11,16#1F,16#00,	// 16#5D
16#00,16#02,16#01,16#02,	// 16#5E
16#20,16#20,16#20,16#20,	// 16#5F
16#00,16#01,16#03,16#00,	// 16#60
16#00,16#18,16#14,16#1C,	// 16#61
16#00,16#1F,16#14,16#08,	// 16#62
16#00,16#08,16#14,16#14,	// 16#63
16#00,16#08,16#14,16#1F,	// 16#64
16#00,16#0C,16#1C,16#14,	// 16#65
16#00,16#04,16#1E,16#05,	// 16#66
16#00,16#2C,16#24,16#3C,	// 16#67
16#00,16#1F,16#04,16#18,	// 16#68
16#00,16#00,16#1D,16#00,	// 16#69
16#00,16#20,16#3D,16#00,	// 16#6A
16#00,16#1F,16#08,16#14,	// 16#6B
16#00,16#00,16#1F,16#00,	// 16#6C
16#00,16#1C,16#0C,16#1C,	// 16#6D
16#00,16#1C,16#04,16#18,	// 16#6E
16#00,16#08,16#14,16#08,	// 16#6F
16#00,16#3C,16#14,16#08,	// 16#70
16#00,16#08,16#14,16#3C,	// 16#71
16#00,16#1C,16#04,16#00,	// 16#72
16#00,16#10,16#1C,16#04,	// 16#73
16#00,16#04,16#1E,16#14,	// 16#74
16#00,16#1C,16#10,16#1C,	// 16#75
16#00,16#0C,16#10,16#0C,	// 16#76
16#00,16#1C,16#18,16#1C,	// 16#77
16#00,16#14,16#08,16#14,	// 16#78
16#00,16#2C,16#10,16#0C,	// 16#79
16#00,16#04,16#1C,16#10,	// 16#7A
16#00,16#04,16#1F,16#11,	// 16#7B
16#00,16#00,16#1F,16#00,	// 16#7C
16#00,16#11,16#1F,16#04,	// 16#7D
16#02,16#01,16#02,16#01,	// 16#7E
16#00,16#0C,16#0A,16#0C,	// 16#7F
16#00,16#2E,16#19,16#09,	// 16#80
16#00,16#0D,16#10,16#1D,	// 16#81
16#00,16#0C,16#1E,16#15,	// 16#82
16#00,16#1A,16#15,16#1E,	// 16#83
16#00,16#19,16#14,16#1D,	// 16#84
16#00,16#19,16#16,16#1C,	// 16#85
16#00,16#18,16#15,16#1C,	// 16#86
16#00,16#2E,16#3A,16#0A,	// 16#87
16#00,16#0E,16#1D,16#16,	// 16#88
16#00,16#0D,16#1C,16#15,	// 16#89
16#00,16#0D,16#1E,16#14,	// 16#8A
16#00,16#01,16#1C,16#01,	// 16#8B
16#00,16#02,16#19,16#02,	// 16#8C
16#00,16#01,16#1A,16#00,	// 16#8D
16#00,16#1D,16#0A,16#1D,	// 16#8E
16#00,16#1C,16#0B,16#1C,	// 16#8F
16#00,16#1C,16#1E,16#15,	// 16#90
16#00,16#18,16#1C,16#0C,	// 16#91
16#00,16#1E,16#1F,16#15,	// 16#92
16#00,16#0A,16#15,16#0A,	// 16#93
16#00,16#09,16#14,16#09,	// 16#94
16#00,16#09,16#16,16#08,	// 16#95
16#00,16#1A,16#11,16#1A,	// 16#96
16#00,16#1D,16#12,16#1C,	// 16#97
16#00,16#2D,16#10,16#0D,	// 16#98
16#00,16#0D,16#12,16#0D,	// 16#99
16#00,16#1D,16#10,16#1D,	// 16#9A
16#00,16#0E,16#1B,16#0A,	// 16#9B
16#00,16#14,16#1E,16#15,	// 16#9C
16#00,16#0B,16#1E,16#0B,	// 16#9D
16#00,16#1E,16#06,16#18,	// 16#9E
16#00,16#10,16#1F,16#05,	// 16#9F
16#00,16#18,16#16,16#1D,	// 16#A0
16#00,16#00,16#1A,16#01,	// 16#A1
16#00,16#1C,16#16,16#1D,	// 16#A2
16#00,16#18,16#12,16#19,	// 16#A3
16#00,16#1D,16#05,16#1D,	// 16#A4
16#00,16#1D,16#09,16#1D,	// 16#A5
16#00,16#16,16#15,16#17,	// 16#A6
16#00,16#12,16#15,16#12,	// 16#A7
16#00,16#08,16#15,16#10,	// 16#A8
16#00,16#0E,16#02,16#02,	// 16#A9
16#02,16#02,16#0E,16#00,	// 16#AA
16#00,16#0B,16#14,16#1A,	// 16#AB
16#00,16#0B,16#0C,16#1A,	// 16#AC
16#00,16#00,16#1D,16#00,	// 16#AD
16#04,16#0A,16#04,16#0A,	// 16#AE
16#0A,16#04,16#0A,16#04,	// 16#AF
16#00,16#15,16#00,16#2A,	// 16#B0
16#2A,16#15,16#2A,16#15,	// 16#B1
16#3F,16#2A,16#3F,16#15,	// 16#B2
16#00,16#00,16#3F,16#00,	// 16#B3
16#04,16#04,16#3F,16#00,	// 16#B4
16#0A,16#0A,16#3F,16#00,	// 16#B5
16#04,16#3F,16#00,16#3F,	// 16#B6
16#04,16#3C,16#04,16#3C,	// 16#B7
16#0A,16#0A,16#3E,16#00,	// 16#B8
16#0A,16#3B,16#00,16#3F,	// 16#B9
16#00,16#3F,16#00,16#3F,	// 16#BA
16#0A,16#3A,16#02,16#3E,	// 16#BB
16#0A,16#0B,16#08,16#0F,	// 16#BC
16#04,16#07,16#04,16#07,	// 16#BD
16#0A,16#0A,16#0F,16#00,	// 16#BE
16#04,16#04,16#3C,16#00,	// 16#BF
16#00,16#00,16#07,16#04,	// 16#C0
16#04,16#04,16#07,16#04,	// 16#C1
16#04,16#04,16#3C,16#04,	// 16#C2
16#00,16#00,16#3F,16#04,	// 16#C3
16#04,16#04,16#04,16#04,	// 16#C4
16#04,16#04,16#3F,16#04,	// 16#C5
16#00,16#00,16#3F,16#0A,	// 16#C6
16#00,16#3F,16#00,16#3F,	// 16#C7
16#00,16#0F,16#08,16#0B,	// 16#C8
16#00,16#3E,16#02,16#3A,	// 16#C9
16#0A,16#0B,16#08,16#0B,	// 16#CA
16#0A,16#3A,16#02,16#3A,	// 16#CB
16#00,16#3F,16#00,16#3B,	// 16#CC
16#0A,16#0A,16#0A,16#0A,	// 16#CD
16#0A,16#3B,16#00,16#3B,	// 16#CE
16#0A,16#0A,16#0B,16#0A,	// 16#CF
16#04,16#07,16#04,16#07,	// 16#D0
16#0A,16#0A,16#3A,16#0A,	// 16#D1
16#04,16#3C,16#04,16#3C,	// 16#D2
16#00,16#07,16#04,16#07,	// 16#D3
16#00,16#00,16#0F,16#0A,	// 16#D4
16#00,16#00,16#3E,16#0A,	// 16#D5
16#00,16#3C,16#04,16#3C,	// 16#D6
16#04,16#3F,16#00,16#3F,	// 16#D7
16#0A,16#0A,16#3B,16#0A,	// 16#D8
16#04,16#04,16#07,16#00,	// 16#D9
16#00,16#00,16#3C,16#04,	// 16#DA
16#3F,16#3F,16#3F,16#3F,	// 16#DB
16#38,16#38,16#38,16#38,	// 16#DC
16#3F,16#3F,16#00,16#00,	// 16#DD
16#00,16#00,16#3F,16#3F,	// 16#DE
16#07,16#07,16#07,16#07,	// 16#DF
16#00,16#1C,16#1C,16#14,	// 16#E0
16#00,16#3E,16#15,16#0A,	// 16#E1
16#00,16#1F,16#01,16#03,	// 16#E2
16#00,16#1F,16#01,16#1F,	// 16#E3
16#00,16#1B,16#15,16#11,	// 16#E4
16#00,16#08,16#14,16#0C,	// 16#E5
16#00,16#3C,16#10,16#1C,	// 16#E6
16#00,16#04,16#1C,16#02,	// 16#E7
16#00,16#15,16#1B,16#15,	// 16#E8
16#00,16#0E,16#15,16#0E,	// 16#E9
16#00,16#1C,16#02,16#1C,	// 16#EA
16#00,16#0A,16#15,16#09,	// 16#EB
16#00,16#1C,16#14,16#1C,	// 16#EC
16#00,16#0E,16#1B,16#0E,	// 16#ED
16#00,16#0E,16#15,16#15,	// 16#EE
16#00,16#1E,16#01,16#1E,	// 16#EF
16#00,16#15,16#15,16#15,	// 16#F0
16#00,16#12,16#17,16#12,	// 16#F1
16#00,16#15,16#15,16#12,	// 16#F2
16#00,16#12,16#15,16#15,	// 16#F3
16#00,16#00,16#3C,16#02,	// 16#F4
16#00,16#10,16#0F,16#00,	// 16#F5
16#00,16#04,16#15,16#04,	// 16#F6
16#14,16#0A,16#14,16#0A,	// 16#F7
16#00,16#02,16#05,16#02,	// 16#F8
16#00,16#04,16#0E,16#04,	// 16#F9
16#00,16#00,16#04,16#00,	// 16#FA
16#00,16#08,16#1F,16#01,	// 16#FB
16#00,16#07,16#01,16#07,	// 16#FC
16#00,16#0D,16#0B,16#00,	// 16#FD
16#00,16#0C,16#0C,16#00,	// 16#FE
16#00,16#00,16#00,16#00 	// 16#FF
];


FONT_5X8:ARRAY[0..255,0..4]OF BYTE :=[
16#00,16#00,16#00,16#00,16#00,	// 16#00
16#1E,16#35,16#31,16#35,16#1E,	// 16#01
16#1E,16#35,16#37,16#35,16#1E,	// 16#02
16#0E,16#1F,16#3E,16#1F,16#0E,	// 16#03
16#08,16#1C,16#7F,16#1C,16#08,	// 16#04
16#18,16#4A,16#7F,16#4A,16#18,	// 16#05
16#1C,16#4E,16#7F,16#4E,16#1C,	// 16#06
16#00,16#00,16#00,16#00,16#00,	// 16#07
16#00,16#00,16#00,16#00,16#00,	// 16#08
16#00,16#00,16#00,16#00,16#00,	// 16#09
16#00,16#00,16#00,16#00,16#00,	// 16#0A
16#38,16#44,16#44,16#47,16#3B,	// 16#0B
16#0E,16#51,16#F1,16#51,16#0E,	// 16#0C
16#00,16#00,16#00,16#00,16#00,	// 16#0D
16#60,16#7E,16#02,16#33,16#3F,	// 16#0E
16#2A,16#1C,16#36,16#1C,16#2A,	// 16#0F
16#3E,16#1C,16#1C,16#08,16#08,	// 16#10
16#08,16#08,16#1C,16#1C,16#3E,	// 16#11
16#00,16#22,16#7F,16#22,16#00,	// 16#12
16#00,16#2E,16#00,16#2E,16#00,	// 16#13
16#06,16#7F,16#01,16#7F,16#00,	// 16#14
16#00,16#4A,16#55,16#29,16#00,	// 16#15
16#00,16#18,16#18,16#18,16#18,	// 16#16
16#00,16#4A,16#5F,16#4A,16#00,	// 16#17
16#00,16#02,16#7F,16#02,16#00,	// 16#18
16#00,16#20,16#7F,16#20,16#00,	// 16#19
16#00,16#08,16#08,16#1C,16#08,	// 16#1A
16#00,16#08,16#1C,16#08,16#08,	// 16#1B
16#00,16#3C,16#20,16#20,16#20,	// 16#1C
16#08,16#1C,16#08,16#1C,16#08,	// 16#1D
16#20,16#38,16#3E,16#38,16#20,	// 16#1E
16#02,16#0E,16#3E,16#0E,16#02,	// 16#1F
16#00,16#00,16#00,16#00,16#00,	// 16#20
16#00,16#00,16#2F,16#00,16#00,	// 16#21
16#00,16#03,16#00,16#03,16#00,	// 16#22
16#34,16#1C,16#36,16#1C,16#16,	// 16#23
16#00,16#26,16#7F,16#32,16#00,	// 16#24
16#32,16#0D,16#1E,16#2C,16#13,	// 16#25
16#18,16#26,16#2D,16#12,16#28,	// 16#26
16#00,16#00,16#03,16#00,16#00,	// 16#27
16#00,16#1C,16#22,16#41,16#41,	// 16#28
16#41,16#41,16#22,16#1C,16#00,	// 16#29
16#00,16#0A,16#05,16#0A,16#00,	// 16#2A
16#00,16#10,16#38,16#10,16#00,	// 16#2B
16#00,16#80,16#60,16#00,16#00,	// 16#2C
16#00,16#08,16#08,16#08,16#00,	// 16#2D
16#00,16#00,16#20,16#00,16#00,	// 16#2E
16#00,16#60,16#18,16#06,16#01,	// 16#2F
16#00,16#1E,16#21,16#21,16#1E,	// 16#30
16#00,16#22,16#3F,16#20,16#00,	// 16#31
16#00,16#31,16#29,16#26,16#00,	// 16#32
16#00,16#25,16#25,16#1A,16#00,	// 16#33
16#00,16#0C,16#0A,16#3F,16#08,	// 16#34
16#00,16#27,16#25,16#19,16#00,	// 16#35
16#00,16#1E,16#25,16#25,16#18,	// 16#36
16#00,16#01,16#39,16#05,16#03,	// 16#37
16#00,16#1A,16#25,16#25,16#1A,	// 16#38
16#00,16#06,16#29,16#29,16#1E,	// 16#39
16#00,16#00,16#24,16#00,16#00,	// 16#3A
16#00,16#80,16#64,16#00,16#00,	// 16#3B
16#00,16#08,16#08,16#14,16#22,	// 16#3C
16#00,16#14,16#14,16#14,16#14,	// 16#3D
16#00,16#22,16#14,16#08,16#08,	// 16#3E
16#00,16#01,16#29,16#05,16#02,	// 16#3F
16#3C,16#42,16#59,16#55,16#5E,	// 16#40
16#30,16#1C,16#12,16#1C,16#30,	// 16#41
16#00,16#3E,16#2A,16#36,16#00,	// 16#42
16#00,16#1C,16#22,16#22,16#22,	// 16#43
16#00,16#3E,16#22,16#22,16#1C,	// 16#44
16#00,16#3E,16#2A,16#2A,16#00,	// 16#45
16#00,16#3E,16#0A,16#0A,16#00,	// 16#46
16#00,16#1C,16#22,16#2A,16#3A,	// 16#47
16#00,16#3E,16#08,16#08,16#3E,	// 16#48
16#00,16#22,16#3E,16#22,16#00,	// 16#49
16#00,16#22,16#22,16#1E,16#00,	// 16#4A
16#00,16#3E,16#08,16#14,16#22,	// 16#4B
16#00,16#3E,16#20,16#20,16#20,	// 16#4C
16#3E,16#04,16#18,16#04,16#3E,	// 16#4D
16#00,16#3E,16#04,16#08,16#3E,	// 16#4E
16#1C,16#22,16#22,16#22,16#1C,	// 16#4F
16#00,16#3E,16#0A,16#0A,16#04,	// 16#50
16#1C,16#22,16#22,16#62,16#9C,	// 16#51
16#00,16#3E,16#0A,16#14,16#20,	// 16#52
16#00,16#24,16#2A,16#12,16#00,	// 16#53
16#02,16#02,16#3E,16#02,16#02,	// 16#54
16#00,16#1E,16#20,16#20,16#1E,	// 16#55
16#00,16#0E,16#30,16#30,16#0E,	// 16#56
16#0E,16#30,16#0C,16#30,16#0E,	// 16#57
16#22,16#14,16#08,16#14,16#22,	// 16#58
16#02,16#04,16#38,16#04,16#02,	// 16#59
16#00,16#32,16#2A,16#2A,16#26,	// 16#5A
16#00,16#00,16#7F,16#41,16#00,	// 16#5B
16#01,16#06,16#18,16#60,16#00,	// 16#5C
16#00,16#41,16#7F,16#00,16#00,	// 16#5D
16#18,16#06,16#01,16#06,16#18,	// 16#5E
16#40,16#40,16#40,16#40,16#40,	// 16#5F
16#00,16#01,16#02,16#00,16#00,	// 16#60
16#00,16#34,16#34,16#38,16#20,	// 16#61
16#00,16#3F,16#24,16#24,16#18,	// 16#62
16#00,16#18,16#24,16#24,16#00,	// 16#63
16#18,16#24,16#24,16#3F,16#00,	// 16#64
16#00,16#18,16#2C,16#28,16#00,	// 16#65
16#00,16#04,16#3E,16#05,16#05,	// 16#66
16#00,16#58,16#54,16#54,16#3C,	// 16#67
16#00,16#3F,16#08,16#04,16#38,	// 16#68
16#00,16#04,16#3D,16#00,16#00,	// 16#69
16#00,16#44,16#44,16#3D,16#00,	// 16#6A
16#00,16#3F,16#08,16#14,16#20,	// 16#6B
16#00,16#01,16#3F,16#00,16#00,	// 16#6C
16#3C,16#08,16#3C,16#08,16#3C,	// 16#6D
16#00,16#3C,16#08,16#04,16#38,	// 16#6E
16#00,16#18,16#24,16#24,16#18,	// 16#6F
16#00,16#7C,16#24,16#24,16#18,	// 16#70
16#18,16#24,16#24,16#7C,16#00,	// 16#71
16#00,16#3C,16#08,16#04,16#00,	// 16#72
16#00,16#28,16#2C,16#14,16#00,	// 16#73
16#00,16#04,16#1E,16#24,16#04,	// 16#74
16#00,16#1C,16#20,16#10,16#3C,	// 16#75
16#00,16#0C,16#30,16#30,16#0C,	// 16#76
16#0C,16#30,16#1C,16#30,16#0C,	// 16#77
16#00,16#24,16#18,16#18,16#24,	// 16#78
16#40,16#4C,16#70,16#30,16#0C,	// 16#79
16#00,16#34,16#2C,16#2C,16#00,	// 16#7A
16#00,16#08,16#36,16#41,16#00,	// 16#7B
16#00,16#00,16#7F,16#00,16#00,	// 16#7C
16#00,16#41,16#36,16#08,16#00,	// 16#7D
16#10,16#08,16#08,16#10,16#08,	// 16#7E
16#00,16#3C,16#22,16#3C,16#00,	// 16#7F
16#00,16#1C,16#A2,16#62,16#22,	// 16#80
16#00,16#1D,16#20,16#10,16#3D,	// 16#81
16#00,16#18,16#2C,16#2A,16#01,	// 16#82
16#00,16#36,16#35,16#39,16#22,	// 16#83
16#00,16#35,16#34,16#39,16#20,	// 16#84
16#01,16#36,16#34,16#38,16#20,	// 16#85
16#00,16#36,16#35,16#3A,16#20,	// 16#86
16#00,16#18,16#A4,16#64,16#00,	// 16#87
16#00,16#1A,16#2D,16#29,16#02,	// 16#88
16#00,16#19,16#2C,16#29,16#00,	// 16#89
16#01,16#1A,16#2C,16#28,16#00,	// 16#8A
16#00,16#05,16#3C,16#01,16#00,	// 16#8B
16#00,16#06,16#3D,16#01,16#02,	// 16#8C
16#01,16#06,16#3C,16#00,16#00,	// 16#8D
16#30,16#1D,16#12,16#1D,16#30,	// 16#8E
16#30,16#1A,16#15,16#1A,16#30,	// 16#8F
16#00,16#3E,16#2A,16#2A,16#01,	// 16#90
16#34,16#14,16#18,16#2C,16#28,	// 16#91
16#30,16#1C,16#12,16#3E,16#2A,	// 16#92
16#02,16#19,16#25,16#26,16#18,	// 16#93
16#00,16#19,16#24,16#24,16#19,	// 16#94
16#01,16#1A,16#24,16#24,16#18,	// 16#95
16#02,16#1D,16#21,16#12,16#3C,	// 16#96
16#00,16#1D,16#22,16#10,16#3C,	// 16#97
16#40,16#4D,16#70,16#30,16#0D,	// 16#98
16#1D,16#22,16#22,16#22,16#1D,	// 16#99
16#01,16#1E,16#20,16#21,16#1E,	// 16#9A
16#00,16#58,16#34,16#2C,16#1A,	// 16#9B
16#10,16#3C,16#2A,16#20,16#00,	// 16#9C
16#5C,16#32,16#2A,16#26,16#1D,	// 16#9D
16#00,16#24,16#18,16#18,16#24,	// 16#9E
16#00,16#48,16#3E,16#09,16#00,	// 16#9F
16#00,16#34,16#34,16#3A,16#21,	// 16#A0
16#00,16#04,16#3C,16#02,16#01,	// 16#A1
16#00,16#18,16#24,16#26,16#19,	// 16#A2
16#00,16#1C,16#20,16#12,16#3D,	// 16#A3
16#00,16#3D,16#09,16#05,16#39,	// 16#A4
16#01,16#3F,16#05,16#09,16#3F,	// 16#A5
16#00,16#1D,16#15,16#1E,16#00,	// 16#A6
16#00,16#0E,16#11,16#0E,16#00,	// 16#A7
16#00,16#40,16#5A,16#20,16#00,	// 16#A8
16#1E,16#21,16#3F,16#37,16#1E,	// 16#A9
16#00,16#08,16#08,16#38,16#00,	// 16#AA
16#21,16#17,16#0C,16#36,16#2D,	// 16#AB
16#21,16#17,16#08,16#16,16#39,	// 16#AC
16#00,16#00,16#74,16#00,16#00,	// 16#AD
16#08,16#14,16#2A,16#14,16#22,	// 16#AE
16#22,16#14,16#2A,16#14,16#08,	// 16#AF
16#55,16#00,16#55,16#00,16#55,	// 16#B0
16#55,16#AA,16#55,16#AA,16#55,	// 16#B1
16#FF,16#55,16#FF,16#55,16#FF,	// 16#B2
16#00,16#00,16#FF,16#00,16#00,	// 16#B3
16#08,16#08,16#FF,16#00,16#00,	// 16#B4
16#30,16#1C,16#12,16#1D,16#30,	// 16#B5
16#30,16#1A,16#15,16#19,16#32,	// 16#B6
16#30,16#1D,16#12,16#1C,16#30,	// 16#B7
16#3E,16#41,16#5D,16#55,16#3E,	// 16#B8
16#14,16#F7,16#00,16#FF,16#00,	// 16#B9
16#00,16#FF,16#00,16#FF,16#00,	// 16#BA
16#14,16#F4,16#04,16#FC,16#00,	// 16#BB
16#14,16#17,16#10,16#1F,16#00,	// 16#BC
16#00,16#1C,16#36,16#14,16#00,	// 16#BD
16#02,16#14,16#38,16#14,16#02,	// 16#BE
16#08,16#08,16#F8,16#00,16#00,	// 16#BF
16#00,16#00,16#0F,16#08,16#08,	// 16#C0
16#08,16#08,16#0F,16#08,16#08,	// 16#C1
16#08,16#08,16#F8,16#08,16#08,	// 16#C2
16#00,16#00,16#FF,16#08,16#08,	// 16#C3
16#08,16#08,16#08,16#08,16#08,	// 16#C4
16#08,16#08,16#FF,16#08,16#08,	// 16#C5
16#02,16#35,16#35,16#3A,16#21,	// 16#C6
16#32,16#19,16#15,16#1A,16#31,	// 16#C7
16#00,16#1F,16#10,16#17,16#14,	// 16#C8
16#00,16#FC,16#04,16#F4,16#14,	// 16#C9
16#14,16#17,16#10,16#17,16#14,	// 16#CA
16#14,16#F4,16#04,16#F4,16#14,	// 16#CB
16#00,16#FF,16#00,16#F7,16#14,	// 16#CC
16#14,16#14,16#14,16#14,16#14,	// 16#CD
16#14,16#F7,16#00,16#F7,16#14,	// 16#CE
16#22,16#1C,16#14,16#1C,16#22,	// 16#CF
16#19,16#25,16#27,16#1D,16#00,	// 16#D0
16#08,16#3E,16#2A,16#22,16#1C,	// 16#D1
16#00,16#3F,16#2B,16#2B,16#00,	// 16#D2
16#01,16#3E,16#2A,16#2A,16#01,	// 16#D3
16#01,16#3E,16#2A,16#2A,16#00,	// 16#D4
16#00,16#04,16#3C,16#00,16#00,	// 16#D5
16#00,16#22,16#3E,16#22,16#01,	// 16#D6
16#00,16#23,16#3F,16#23,16#00,	// 16#D7
16#01,16#22,16#3E,16#22,16#01,	// 16#D8
16#08,16#08,16#0F,16#00,16#00,	// 16#D9
16#00,16#00,16#F8,16#08,16#08,	// 16#DA
16#FF,16#FF,16#FF,16#FF,16#FF,	// 16#DB
16#F0,16#F0,16#F0,16#F0,16#F0,	// 16#DC
16#00,16#00,16#E7,16#00,16#00,	// 16#DD
16#01,16#22,16#3E,16#22,16#00,	// 16#DE
16#0F,16#0F,16#0F,16#0F,16#0F,	// 16#DF
16#1C,16#22,16#22,16#22,16#1D,	// 16#E0
16#00,16#3E,16#01,16#2E,16#10,	// 16#E1
16#1C,16#23,16#23,16#23,16#1C,	// 16#E2
16#1D,16#22,16#22,16#22,16#1C,	// 16#E3
16#02,16#19,16#25,16#26,16#19,	// 16#E4
16#1D,16#23,16#23,16#23,16#1C,	// 16#E5
16#00,16#7C,16#20,16#10,16#3C,	// 16#E6
16#00,16#7F,16#24,16#24,16#18,	// 16#E7
16#00,16#3E,16#14,16#14,16#08,	// 16#E8
16#1E,16#20,16#20,16#1E,16#01,	// 16#E9
16#00,16#1F,16#21,16#21,16#1F,	// 16#EA
16#01,16#1E,16#20,16#20,16#1E,	// 16#EB
16#40,16#4C,16#30,16#32,16#0D,	// 16#EC
16#02,16#04,16#3A,16#05,16#02,	// 16#ED
16#01,16#01,16#01,16#01,16#01,	// 16#EE
16#00,16#00,16#02,16#01,16#00,	// 16#EF
16#00,16#08,16#08,16#08,16#00,	// 16#F0
16#00,16#28,16#3C,16#28,16#00,	// 16#F1
16#A0,16#A0,16#A0,16#A0,16#A0,	// 16#F2
16#2B,16#1F,16#08,16#16,16#39,	// 16#F3
16#06,16#7F,16#01,16#7F,16#00,	// 16#F4
16#00,16#4A,16#55,16#29,16#00,	// 16#F5
16#00,16#08,16#2A,16#08,16#00,	// 16#F6
16#00,16#80,16#40,16#00,16#00,	// 16#F7
16#00,16#06,16#09,16#09,16#06,	// 16#F8
16#00,16#01,16#00,16#01,16#00,	// 16#F9
16#00,16#00,16#08,16#00,16#00,	// 16#FA
16#00,16#11,16#1F,16#10,16#00,	// 16#FB
16#00,16#15,16#15,16#0A,16#00,	// 16#FC
16#00,16#19,16#15,16#12,16#00,	// 16#FD
16#00,16#3C,16#3C,16#3C,16#3C,	// 16#FE
16#00,16#00,16#00,16#00,16#00 	// 16#FF
];


